C01810=1014.320,152.108,374.636,166.710,56.034,160.285
C01811=1014.316,151.858,374.655,166.706,56.046,160.287
C01812=1014.312,151.609,374.675,166.703,56.058,160.288
C01813=1014.308,151.360,374.694,166.700,56.069,160.290
C01814=1014.304,151.110,374.713,166.697,56.080,160.291
C01815=1014.299,150.861,374.732,166.693,56.091,160.293
C01816=1014.295,150.612,374.751,166.690,56.103,160.294
C01817=1014.291,150.363,374.771,166.686,56.115,160.296
C01818=1014.287,150.113,374.789,166.683,56.126,160.297
C01819=1014.283,149.864,374.809,166.680,56.138,160.299
C01820=1014.279,149.615,374.827,166.676,56.149,160.300
C01821=1014.275,149.366,374.847,166.673,56.160,160.302
C01822=1014.270,149.116,374.865,166.670,56.172,160.303
C01823=1014.266,148.867,374.884,166.667,56.183,160.305
C01824=1014.262,148.618,374.903,166.663,56.194,160.306
C01825=1014.257,148.369,374.923,166.659,56.206,160.308
C01826=1014.253,148.119,374.941,166.656,56.218,160.309
C01827=1014.249,147.870,374.961,166.654,56.229,160.311
C01828=1014.245,147.621,374.979,166.650,56.240,160.312
C01829=1014.241,147.372,374.999,166.646,56.252,160.314
C01830=1014.237,147.122,375.017,166.643,56.263,160.315
C01831=1014.233,146.873,375.036,166.640,56.275,160.317
C01832=1014.229,146.624,375.056,166.636,56.286,160.318
C01833=1014.224,146.374,375.074,166.633,56.297,160.320
C01834=1014.220,146.126,375.093,166.630,56.309,160.321
C01835=1014.216,145.876,375.112,166.627,56.321,160.323
C01836=1014.212,145.627,375.130,166.623,56.332,160.324
C01837=1014.208,145.378,375.150,166.620,56.343,160.326
C01838=1014.204,145.128,375.169,166.617,56.355,160.327
C01839=1014.199,144.879,375.186,166.614,56.366,160.329
C01840=1014.195,144.630,375.205,166.610,56.378,160.330
C01841=1014.191,144.381,375.225,166.607,56.389,160.332
C01842=1014.186,144.131,375.243,166.603,56.401,160.333
C01843=1014.182,143.882,375.262,166.601,56.412,160.335
C01844=1014.178,143.633,375.279,166.598,56.424,160.336
C01845=1014.174,143.384,375.299,166.594,56.435,160.338
C01846=1014.170,143.134,375.318,166.591,56.446,160.339
C01847=1014.165,142.885,375.336,166.587,56.458,160.341
C01848=1014.161,142.636,375.354,166.585,56.469,160.342
C01849=1014.157,142.386,375.373,166.582,56.481,160.344
C01850=1014.153,142.137,375.391,166.578,56.492,160.345
C01851=1014.148,141.888,375.411,166.575,56.504,160.347
C01852=1014.145,141.639,375.429,166.572,56.515,160.349
C01853=1014.140,141.390,375.447,166.568,56.526,160.350
C01854=1014.136,141.140,375.466,166.565,56.538,160.351
C01855=1014.132,140.890,375.485,166.562,56.550,160.353
C01856=1014.128,140.642,375.502,166.560,56.561,160.355
C01857=1014.124,140.392,375.521,166.556,56.572,160.356
C01858=1014.119,140.143,375.541,166.553,56.584,160.357
C01859=1014.115,139.894,375.558,166.550,56.595,160.359
C01860=1014.111,139.645,375.577,166.546,56.606,160.360
C01861=1014.107,139.395,375.596,166.543,56.618,160.362
C01862=1014.102,139.146,375.614,166.540,56.629,160.364
C01863=1014.098,138.866,375.635,166.537,56.642,160.365
C01864=1014.094,138.586,375.656,166.533,56.654,160.367
C01865=1014.088,138.306,375.677,166.529,56.667,160.368
C01866=1014.085,138.026,375.697,166.526,56.680,160.370
C01867=1014.080,137.776,375.715,166.523,56.691,160.372
C01868=1014.076,137.527,375.734,166.520,56.703,160.373
C01869=1014.072,137.278,375.752,166.516,56.714,160.375
C01870=1014.068,137.028,375.770,166.514,56.725,160.376
C01871=1014.063,136.779,375.789,166.511,56.737,160.378
C01872=1014.060,136.530,375.807,166.507,56.748,160.379
C01873=1014.055,136.281,375.825,166.505,56.759,160.381
C01874=1014.051,136.031,375.844,166.502,56.771,160.383
C01875=1014.047,135.782,375.862,166.498,56.782,160.384
C01876=1014.043,135.533,375.881,166.496,56.794,160.386
C01877=1014.038,135.283,375.899,166.493,56.805,160.387
C01878=1014.034,135.034,375.917,166.489,56.817,160.388
C01879=1014.030,134.784,375.935,166.487,56.828,160.390
C01880=1014.025,134.535,375.953,166.483,56.839,160.391
C01881=1014.022,134.286,375.971,166.480,56.851,160.393
C01882=1014.017,134.037,375.989,166.478,56.862,160.395
C01883=1014.013,133.788,376.007,166.474,56.873,160.396
C01884=1014.009,133.538,376.026,166.471,56.885,160.398
C01885=1014.004,133.288,376.043,166.469,56.896,160.399
C01886=1014.001,133.039,376.062,166.465,56.907,160.401
C01887=1013.996,132.790,376.080,166.463,56.919,160.402
C01888=1013.992,132.541,376.098,166.459,56.930,160.404
C01889=1013.988,132.291,376.116,166.456,56.942,160.405
C01890=1013.984,132.043,376.133,166.454,56.953,160.407
C01891=1013.979,131.793,376.152,166.450,56.964,160.408
C01892=1013.975,131.544,376.170,166.448,56.975,160.410
C01893=1013.971,131.295,376.188,166.444,56.987,160.411
C01894=1013.967,131.045,376.206,166.441,56.998,160.413
C01895=1013.963,130.796,376.224,166.438,57.009,160.414
C01896=1013.958,130.547,376.242,166.435,57.021,160.416
C01897=1013.955,130.298,376.261,166.432,57.032,160.418
C01898=1013.950,130.048,376.278,166.429,57.043,160.419
C01899=1013.946,129.798,376.297,166.427,57.054,160.421
C01900=1013.942,129.549,376.315,166.424,57.066,160.422
C01901=1013.938,129.299,376.332,166.421,57.077,160.424
C01902=1013.933,129.051,376.350,166.418,57.088,160.425
C01903=1013.929,128.801,376.367,166.415,57.100,160.427
C01904=1013.925,128.552,376.385,166.412,57.111,160.428
C01905=1013.921,128.302,376.403,166.409,57.123,160.430
C01906=1013.917,128.053,376.421,166.406,57.135,160.431
C01907=1013.912,127.803,376.438,166.403,57.145,160.433
C01908=1013.908,127.555,376.456,166.400,57.157,160.435
C01909=1013.904,127.305,376.474,166.397,57.168,160.436
C01910=1013.899,127.056,376.491,166.394,57.180,160.438
C01911=1013.895,126.806,376.509,166.391,57.192,160.439
C01912=1013.891,126.557,376.526,166.389,57.202,160.441
C01913=1013.886,126.307,376.544,166.386,57.214,160.442
C01914=1013.882,126.058,376.561,166.383,57.225,160.444
C01915=1013.878,125.809,376.579,166.380,57.237,160.445
C01916=1013.874,125.559,376.596,166.377,57.247,160.447
C01917=1013.869,125.310,376.614,166.374,57.259,160.448
C01918=1013.865,125.061,376.632,166.371,57.270,160.450
C01919=1013.861,124.811,376.649,166.369,57.282,160.452
C01920=1013.856,124.562,376.667,166.366,57.294,160.453
C01921=1013.852,124.312,376.684,166.363,57.304,160.455
C01922=1013.848,124.064,376.702,166.360,57.316,160.456
C01923=1013.843,123.814,376.719,166.357,57.327,160.458
C01924=1013.839,123.564,376.737,166.354,57.338,160.459
C01925=1013.835,123.315,376.755,166.352,57.350,160.461
C01926=1013.831,123.066,376.772,166.348,57.361,160.462
C01927=1013.826,122.786,376.791,166.346,57.373,160.464
C01928=1013.821,122.506,376.811,166.342,57.386,160.466
C01929=1013.817,122.226,376.831,166.340,57.399,160.468
C01930=1013.812,121.946,376.850,166.336,57.411,160.469
C01931=1013.807,121.697,376.868,166.334,57.423,160.471
C01932=1013.803,121.447,376.885,166.330,57.434,160.472
C01933=1013.799,121.197,376.903,166.328,57.445,160.474
C01934=1013.795,120.949,376.920,166.326,57.456,160.475
C01935=1013.791,120.699,376.937,166.322,57.467,160.477
C01936=1013.786,120.449,376.955,166.319,57.478,160.478
C01937=1013.782,120.201,376.973,166.316,57.490,160.480
C01938=1013.778,119.952,376.990,166.314,57.501,160.481
C01939=1013.774,119.702,377.007,166.311,57.511,160.483
C01940=1013.770,119.453,377.025,166.308,57.523,160.485
C01941=1013.765,119.203,377.042,166.306,57.534,160.486
C01942=1013.761,118.954,377.060,166.302,57.545,160.487
C01943=1013.757,118.704,377.077,166.300,57.557,160.489
C01944=1013.753,118.455,377.095,166.298,57.568,160.491
C01945=1013.749,118.206,377.112,166.294,57.579,160.492
C01946=1013.745,117.956,377.129,166.292,57.589,160.493
C01947=1013.740,117.707,377.146,166.290,57.601,160.495
C01948=1013.736,117.458,377.164,166.286,57.612,160.497
C01949=1013.732,117.209,377.181,166.284,57.623,160.498
C01950=1013.728,116.959,377.199,166.281,57.634,160.500
C01951=1013.724,116.709,377.216,166.279,57.645,160.501
C01952=1013.720,116.461,377.234,166.276,57.656,160.503
C01953=1013.715,116.211,377.251,166.273,57.667,160.504
C01954=1013.712,115.961,377.269,166.271,57.678,160.506
C01955=1013.708,115.712,377.286,166.267,57.689,160.507
C01956=1013.704,115.462,377.303,166.265,57.700,160.509
C01957=1013.700,115.213,377.321,166.263,57.711,160.510
C01958=1013.696,114.964,377.338,166.261,57.722,160.512
C01959=1013.691,114.714,377.356,166.257,57.733,160.513
C01960=1013.687,114.465,377.373,166.255,57.744,160.515
C01961=1013.683,114.215,377.390,166.252,57.755,160.516
C01962=1013.680,113.966,377.407,166.250,57.766,160.518
C01963=1013.675,113.717,377.425,166.247,57.777,160.519
C01964=1013.671,113.468,377.442,166.244,57.788,160.521
C01965=1013.667,113.218,377.459,166.241,57.799,160.522
C01966=1013.663,112.969,377.476,166.239,57.809,160.524
C01967=1013.659,112.719,377.494,166.237,57.821,160.526
C01968=1013.655,112.470,377.511,166.235,57.832,160.527
C01969=1013.651,112.221,377.528,166.232,57.843,160.529
C01970=1013.647,111.972,377.546,166.229,57.854,160.530
C01971=1013.642,111.722,377.563,166.226,57.865,160.532
C01972=1013.638,111.473,377.579,166.224,57.875,160.533
C01973=1013.634,111.224,377.597,166.221,57.886,160.535
C01974=1013.630,110.973,377.613,166.218,57.897,160.536
C01975=1013.625,110.724,377.630,166.215,57.908,160.537
C01976=1013.621,110.475,377.647,166.213,57.919,160.539
C01977=1013.617,110.226,377.664,166.211,57.930,160.541
C01978=1013.613,109.977,377.680,166.208,57.941,160.542
C01979=1013.608,109.727,377.698,166.205,57.953,160.544
C01980=1013.604,109.477,377.715,166.203,57.964,160.545
C01981=1013.600,109.228,377.732,166.201,57.974,160.547
C01982=1013.596,108.979,377.749,166.198,57.985,160.548
C01983=1013.591,108.729,377.766,166.196,57.996,160.550
C01984=1013.587,108.480,377.782,166.192,58.007,160.551
C01985=1013.583,108.230,377.799,166.190,58.018,160.553
C01986=1013.579,107.981,377.815,166.188,58.029,160.554
C01987=1013.575,107.732,377.832,166.185,58.040,160.556
C01988=1013.570,107.482,377.849,166.183,58.051,160.557
C01989=1013.566,107.233,377.866,166.179,58.062,160.559
C01990=1013.561,106.984,377.882,166.177,58.073,160.560
C01991=1013.557,106.704,377.901,166.175,58.085,160.562
C01992=1013.552,106.423,377.919,166.172,58.097,160.564
C01993=1013.547,106.144,377.939,166.169,58.109,160.566
C01994=1013.542,105.864,377.957,166.166,58.121,160.567
C01995=1013.538,105.615,377.974,166.163,58.133,160.569
C01996=1013.534,105.365,377.990,166.161,58.144,160.570
C01997=1013.530,105.116,378.007,166.158,58.154,160.572
C01998=1013.525,104.867,378.024,166.156,58.165,160.573
C01999=1013.522,104.617,378.040,166.154,58.176,160.575
C02000=1013.517,104.367,378.057,166.151,58.187,160.576
C02001=1013.513,104.118,378.074,166.149,58.198,160.578
C02002=1013.508,103.869,378.090,166.147,58.209,160.579
C02003=1013.505,103.619,378.107,166.144,58.220,160.581
C02004=1013.500,103.370,378.123,166.141,58.231,160.582
C02005=1013.496,103.121,378.140,166.139,58.242,160.584
C02006=1013.492,102.871,378.156,166.136,58.253,160.586
C02007=1013.488,102.622,378.173,166.133,58.263,160.587
C02008=1013.483,102.372,378.189,166.131,58.274,160.588
C02009=1013.479,102.123,378.206,166.129,58.285,160.590
C02010=1013.475,101.874,378.223,166.126,58.295,160.591
C02011=1013.471,101.624,378.239,166.124,58.306,160.593
C02012=1013.467,101.374,378.256,166.122,58.317,160.595
C02013=1013.463,101.125,378.273,166.119,58.327,160.596
C02014=1013.459,100.876,378.289,166.117,58.338,160.597
C02015=1013.454,100.627,378.306,166.114,58.349,160.599
C02016=1013.450,100.377,378.323,166.112,58.360,160.601
C02017=1013.446,100.128,378.338,166.109,58.370,160.602
C02018=1013.442,99.878,378.356,166.107,58.381,160.603
C02019=1013.437,99.628,378.372,166.106,58.391,160.605
C02020=1013.434,99.379,378.389,166.103,58.402,160.607
C02021=1013.429,99.130,378.405,166.100,58.412,160.608
C02022=1013.425,98.880,378.422,166.098,58.423,160.610
C02023=1013.421,98.631,378.438,166.096,58.434,160.611
C02024=1013.416,98.382,378.454,166.093,58.444,160.612
C02025=1013.412,98.132,378.470,166.091,58.455,160.614
C02026=1013.408,97.883,378.487,166.088,58.466,160.616
C02027=1013.404,97.633,378.502,166.086,58.477,160.617
C02028=1013.399,97.384,378.519,166.084,58.488,160.619
C02029=1013.395,97.135,378.535,166.081,58.498,160.620
C02030=1013.391,96.885,378.551,166.079,58.509,160.622
C02031=1013.387,96.636,378.568,166.077,58.520,160.623
C02032=1013.383,96.386,378.583,166.074,58.530,160.624
C02033=1013.378,96.137,378.599,166.072,58.541,160.626
C02034=1013.374,95.888,378.616,166.069,58.552,160.628
C02035=1013.370,95.638,378.632,166.067,58.563,160.629
C02036=1013.366,95.388,378.648,166.064,58.573,160.630
C02037=1013.361,95.139,378.664,166.062,58.584,160.632
C02038=1013.357,94.890,378.680,166.059,58.594,160.633
C02039=1013.353,94.640,378.696,166.058,58.605,160.635
C02040=1013.349,94.391,378.713,166.056,58.616,160.637
C02041=1013.344,94.141,378.729,166.053,58.626,160.638
C02042=1013.340,93.892,378.744,166.051,58.637,160.639
C02043=1013.335,93.643,378.761,166.048,58.647,160.641
C02044=1013.331,93.393,378.777,166.046,58.658,160.642
C02045=1013.328,93.143,378.793,166.043,58.669,160.644
C02046=1013.323,92.894,378.809,166.042,58.679,160.645
C02047=1013.319,92.645,378.825,166.040,58.689,160.647
C02048=1013.314,92.395,378.841,166.037,58.700,160.648
C02049=1013.310,92.146,378.857,166.035,58.711,160.650
C02050=1013.306,91.896,378.874,166.032,58.721,160.651
C02051=1013.302,91.647,378.890,166.031,58.731,160.653
C02052=1013.298,91.397,378.905,166.028,58.742,160.654
C02053=1013.293,91.148,378.922,166.025,58.752,160.655
C02054=1013.289,90.899,378.938,166.023,58.763,160.657
C02055=1013.285,90.619,378.956,166.021,58.774,160.659
C02056=1013.279,90.339,378.974,166.018,58.786,160.660
C02057=1013.275,90.060,378.992,166.015,58.798,160.662
C02058=1013.270,89.781,379.010,166.013,58.809,160.664
C02059=1013.266,89.531,379.025,166.011,58.819,160.665
C02060=1013.262,89.282,379.042,166.008,58.830,160.667
C02061=1013.258,89.032,379.058,166.007,58.840,160.668
C02062=1013.254,88.782,379.073,166.004,58.850,160.669
C02063=1013.249,88.533,379.090,166.002,58.861,160.671
C02064=1013.245,88.284,379.106,166.000,58.871,160.673
C02065=1013.240,88.034,379.121,165.998,58.882,160.674
C02066=1013.236,87.785,379.137,165.995,58.892,160.675
C02067=1013.232,87.535,379.153,165.992,58.902,160.677
C02068=1013.227,87.286,379.169,165.991,58.913,160.679
C02069=1013.223,87.036,379.184,165.989,58.923,160.680
C02070=1013.219,86.787,379.200,165.986,58.934,160.681
C02071=1013.214,86.538,379.215,165.984,58.944,160.683
C02072=1013.210,86.288,379.231,165.982,58.954,160.684
C02073=1013.206,86.039,379.247,165.980,58.965,160.686
C02074=1013.201,85.789,379.262,165.977,58.975,160.687
C02075=1013.197,85.539,379.278,165.975,58.985,160.689
C02076=1013.193,85.290,379.294,165.973,58.996,160.690
C02077=1013.189,85.040,379.309,165.971,59.006,160.692
C02078=1013.185,84.790,379.325,165.969,59.016,160.693
C02079=1013.180,84.542,379.340,165.966,59.026,160.694
C02080=1013.176,84.292,379.355,165.964,59.037,160.696
C02081=1013.172,84.042,379.371,165.962,59.047,160.697
C02082=1013.167,83.793,379.387,165.960,59.057,160.699
C02083=1013.163,83.543,379.403,165.958,59.067,160.700
C02084=1013.159,83.294,379.418,165.955,59.077,160.702
C02085=1013.154,83.044,379.434,165.954,59.087,160.703
C02086=1013.151,82.795,379.450,165.952,59.098,160.705
C02087=1013.146,82.546,379.465,165.949,59.108,160.706
C02088=1013.141,82.296,379.480,165.947,59.118,160.708
C02089=1013.137,82.047,379.496,165.945,59.128,160.709
C02090=1013.133,81.797,379.512,165.943,59.138,160.710
C02091=1013.129,81.548,379.527,165.940,59.149,160.712
C02092=1013.125,81.298,379.542,165.939,59.158,160.713
C02093=1013.121,81.049,379.558,165.936,59.169,160.714
C02094=1013.116,80.799,379.574,165.934,59.178,160.716
C02095=1013.111,80.550,379.589,165.932,59.189,160.717
C02096=1013.107,80.300,379.605,165.930,59.199,160.719
C02097=1013.103,80.051,379.620,165.927,59.209,160.720
C02098=1013.099,79.802,379.636,165.926,59.219,160.722
C02099=1013.095,79.551,379.651,165.923,59.229,160.723
C02100=1013.091,79.302,379.667,165.921,59.239,160.724
C02101=1013.086,79.052,379.683,165.920,59.249,160.726
C02102=1013.083,78.803,379.698,165.917,59.259,160.727
C02103=1013.078,78.554,379.713,165.915,59.269,160.729
C02104=1013.073,78.305,379.729,165.913,59.279,160.730
C02105=1013.069,78.055,379.745,165.911,59.289,160.732
C02106=1013.066,77.806,379.760,165.910,59.299,160.733
C02107=1013.061,77.556,379.775,165.906,59.308,160.734
C02108=1013.057,77.306,379.791,165.905,59.318,160.736
C02109=1013.053,77.057,379.807,165.903,59.328,160.737
C02110=1013.049,76.807,379.822,165.900,59.338,160.739
C02111=1013.044,76.558,379.837,165.899,59.348,160.740
C02112=1013.040,76.308,379.852,165.897,59.358,160.742
C02113=1013.036,76.059,379.868,165.894,59.367,160.743
C02114=1013.031,75.809,379.883,165.892,59.377,160.744
C02115=1013.027,75.560,379.898,165.891,59.387,160.746
C02116=1013.023,75.311,379.914,165.888,59.397,160.747
C02117=1013.018,75.061,379.928,165.887,59.407,160.749
C02118=1013.014,74.811,379.944,165.884,59.418,160.750
C02119=1013.010,74.572,379.958,165.882,59.427,160.751
C02120=1013.006,74.331,379.973,165.880,59.436,160.752
C02121=1013.002,74.092,379.987,165.878,59.446,160.754
C02122=1012.997,73.852,380.002,165.876,59.455,160.755
C02123=1012.994,73.612,380.017,165.874,59.465,160.757
C02124=1012.989,73.372,380.031,165.872,59.474,160.758
C02125=1012.985,73.133,380.045,165.870,59.484,160.759
C02126=1012.981,72.892,380.060,165.868,59.493,160.761
C02127=1012.977,72.643,380.075,165.867,59.503,160.762
C02128=1012.973,72.393,380.090,165.865,59.512,160.763
C02129=1012.968,72.144,380.105,165.862,59.522,160.765
C02130=1012.964,71.895,380.121,165.860,59.532,160.766
C02131=1012.959,71.645,380.135,165.858,59.541,160.767
C02132=1012.955,71.396,380.151,165.857,59.551,160.769
C02133=1012.951,71.147,380.165,165.854,59.560,160.770
C02134=1012.947,70.897,380.181,165.852,59.570,160.771
C02135=1012.943,70.647,380.196,165.850,59.580,160.773
C02136=1012.938,70.398,380.211,165.848,59.589,160.774
C02137=1012.934,70.148,380.226,165.847,59.599,160.776
C02138=1012.929,69.899,380.241,165.844,59.608,160.777
C02139=1012.926,69.649,380.256,165.843,59.618,160.779
C02140=1012.921,69.400,380.271,165.840,59.628,160.780
C02141=1012.917,69.150,380.286,165.838,59.638,160.781
C02142=1012.912,68.901,380.301,165.836,59.647,160.782
C02143=1012.908,68.651,380.316,165.835,59.657,160.784
C02144=1012.903,68.402,380.331,165.832,59.666,160.785
C02145=1012.900,68.152,380.346,165.830,59.675,160.786
C02146=1012.895,67.903,380.361,165.829,59.685,160.788
C02147=1012.891,67.653,380.376,165.827,59.694,160.789
C02148=1012.887,67.404,380.390,165.825,59.704,160.791
C02149=1012.882,67.154,380.406,165.823,59.713,160.792
C02150=1012.878,66.904,380.420,165.821,59.723,160.793
C02151=1012.874,66.655,380.435,165.818,59.733,160.794
C02152=1012.869,66.405,380.450,165.816,59.742,160.796
C02153=1012.865,66.156,380.464,165.815,59.752,160.797
C02154=1012.861,65.906,380.479,165.812,59.761,160.798
C02155=1012.856,65.657,380.494,165.810,59.770,160.800
C02156=1012.853,65.407,380.509,165.809,59.780,160.801
C02157=1012.848,65.157,380.523,165.807,59.789,160.802
C02158=1012.843,64.909,380.538,165.805,59.798,160.804
C02159=1012.839,64.659,380.553,165.803,59.808,160.805
C02160=1012.835,64.409,380.568,165.801,59.817,160.806
C02161=1012.830,64.160,380.583,165.799,59.826,160.808
C02162=1012.826,63.910,380.598,165.797,59.836,160.809
C02163=1012.822,63.661,380.612,165.795,59.845,160.811
C02164=1012.817,63.411,380.626,165.793,59.855,160.812
C02165=1012.813,63.161,380.642,165.791,59.864,160.813
C02166=1012.809,62.912,380.656,165.790,59.873,160.814
C02167=1012.804,62.662,380.671,165.788,59.882,160.816
C02168=1012.801,62.413,380.685,165.786,59.891,160.817
C02169=1012.796,62.163,380.700,165.784,59.901,160.818
C02170=1012.791,61.913,380.714,165.782,59.910,160.820
C02171=1012.787,61.664,380.728,165.780,59.919,160.821
C02172=1012.782,61.414,380.743,165.778,59.928,160.822
C02173=1012.778,61.165,380.757,165.777,59.938,160.824
C02174=1012.773,60.915,380.772,165.775,59.947,160.825
C02175=1012.769,60.666,380.786,165.773,59.957,160.826
C02176=1012.764,60.416,380.800,165.770,59.966,160.827
C02177=1012.760,60.167,380.815,165.768,59.975,160.829
C02178=1012.755,59.917,380.829,165.766,59.984,160.830
C02179=1012.732,71.816,379.715,165.827,59.747,160.800
C02180=1012.736,72.066,379.701,165.829,59.737,160.799
C02181=1012.741,72.316,379.685,165.831,59.728,160.797
C02182=1012.745,72.565,379.671,165.833,59.719,160.796
C02183=1012.749,72.814,379.655,165.834,59.709,160.795
C02184=1012.753,73.059,379.641,165.837,59.700,160.793
C02185=1012.757,73.305,379.627,165.839,59.691,160.792
C02186=1012.762,73.551,379.612,165.840,59.681,160.791
C02187=1012.765,73.796,379.597,165.842,59.672,160.789
C02188=1012.770,74.042,379.582,165.844,59.662,160.788
C02189=1012.774,74.286,379.567,165.846,59.653,160.787
C02190=1012.778,74.532,379.552,165.848,59.644,160.785
C02191=1012.783,74.778,379.537,165.851,59.633,160.784
C02192=1012.787,75.026,379.522,165.853,59.624,160.783
C02193=1012.791,75.276,379.507,165.854,59.614,160.781
C02194=1012.796,75.526,379.492,165.856,59.604,160.780
C02195=1012.799,75.775,379.477,165.858,59.595,160.778
C02196=1012.803,76.025,379.461,165.861,59.585,160.777
C02197=1012.809,76.274,379.446,165.863,59.576,160.776
C02198=1012.812,76.524,379.431,165.864,59.566,160.774
C02199=1012.816,76.773,379.416,165.866,59.556,160.773
C02200=1012.820,77.024,379.401,165.868,59.547,160.772
C02201=1012.825,77.273,379.385,165.871,59.537,160.770
C02202=1012.829,77.522,379.370,165.873,59.528,160.769
C02203=1012.833,77.771,379.354,165.874,59.518,160.767
C02204=1012.837,78.021,379.339,165.876,59.508,160.766
C02205=1012.842,78.271,379.323,165.879,59.498,160.765
C02206=1012.845,78.520,379.308,165.881,59.488,160.763
C02207=1012.850,78.769,379.292,165.882,59.478,160.762
C02208=1012.854,79.020,379.277,165.884,59.469,160.761
C02209=1012.858,79.268,379.262,165.887,59.459,160.759
C02210=1012.862,79.518,379.247,165.889,59.449,160.758
C02211=1012.867,79.767,379.231,165.890,59.439,160.756
C02212=1012.871,80.017,379.215,165.894,59.430,160.755
C02213=1012.874,80.266,379.200,165.895,59.420,160.754
C02214=1012.879,80.516,379.185,165.897,59.410,160.752
C02215=1012.883,80.766,379.169,165.899,59.400,160.751
C02216=1012.887,81.015,379.153,165.901,59.390,160.749
C02217=1012.891,81.264,379.138,165.902,59.380,160.748
C02218=1012.896,81.513,379.122,165.906,59.371,160.747
C02219=1012.900,81.764,379.107,165.907,59.361,160.745
C02220=1012.904,82.013,379.092,165.910,59.350,160.744
C02221=1012.908,82.262,379.076,165.911,59.341,160.742
C02222=1012.912,82.512,379.060,165.913,59.331,160.741
C02223=1012.917,82.761,379.045,165.916,59.320,160.740
C02224=1012.921,83.011,379.029,165.917,59.311,160.738
C02225=1012.925,83.261,379.014,165.920,59.300,160.737
C02226=1012.929,83.509,378.999,165.922,59.290,160.735
C02227=1012.934,83.759,378.983,165.924,59.280,160.734
C02228=1012.938,84.009,378.968,165.926,59.270,160.732
C02229=1012.942,84.258,378.952,165.928,59.260,160.731
C02230=1012.947,84.508,378.936,165.930,59.250,160.729
C02231=1012.950,84.757,378.921,165.933,59.240,160.728
C02232=1012.954,85.007,378.906,165.934,59.230,160.727
C02233=1012.959,85.256,378.890,165.937,59.220,160.725
C02234=1012.964,85.506,378.875,165.939,59.210,160.724
C02235=1012.968,85.755,378.859,165.941,59.200,160.722
C02236=1012.972,86.005,378.843,165.942,59.189,160.721
C02237=1012.976,86.254,378.828,165.945,59.179,160.719
C02238=1012.980,86.503,378.812,165.948,59.169,160.718
C02239=1012.985,86.753,378.796,165.949,59.159,160.716
C02240=1012.989,87.002,378.780,165.952,59.149,160.715
C02241=1012.993,87.252,378.765,165.954,59.139,160.714
C02242=1012.997,87.502,378.749,165.956,59.128,160.712
C02243=1013.002,87.750,378.734,165.958,59.117,160.711
C02244=1013.006,88.000,378.718,165.960,59.108,160.709
C02245=1013.010,88.250,378.703,165.963,59.097,160.708
C02246=1013.015,88.500,378.687,165.965,59.086,160.706
C02247=1013.019,88.749,378.672,165.966,59.077,160.705
C02248=1013.023,88.998,378.655,165.969,59.066,160.703
C02249=1013.027,89.248,378.639,165.972,59.056,160.702
C02250=1013.031,89.498,378.623,165.974,59.046,160.701
C02251=1013.035,89.746,378.608,165.976,59.035,160.699
C02252=1013.041,90.026,378.590,165.978,59.024,160.697
C02253=1013.045,90.306,378.571,165.981,59.013,160.696
C02254=1013.049,90.585,378.554,165.982,59.001,160.694
C02255=1013.054,90.864,378.536,165.986,58.990,160.693
C02256=1013.058,91.114,378.520,165.988,58.979,160.691
C02257=1013.062,91.363,378.504,165.989,58.969,160.689
C02258=1013.067,91.613,378.488,165.992,58.959,160.688
C02259=1013.070,91.862,378.471,165.995,58.948,160.687
C02260=1013.075,92.112,378.455,165.996,58.938,160.685
C02261=1013.078,92.360,378.440,165.999,58.928,160.684
C02262=1013.083,92.610,378.424,166.001,58.917,160.682
C02263=1013.087,92.860,378.408,166.004,58.906,160.681
C02264=1013.091,93.109,378.391,166.005,58.897,160.679
C02265=1013.095,93.358,378.376,166.008,58.886,160.678
C02266=1013.100,93.608,378.360,166.010,58.876,160.676
C02267=1013.104,93.858,378.344,166.013,58.865,160.675
C02268=1013.108,94.107,378.328,166.014,58.855,160.673
C02269=1013.112,94.356,378.311,166.017,58.845,160.672
C02270=1013.116,94.606,378.295,166.019,58.834,160.670
C02271=1013.121,94.856,378.280,166.022,58.823,160.669
C02272=1013.125,95.105,378.263,166.024,58.812,160.668
C02273=1013.130,95.354,378.247,166.026,58.803,160.666
C02274=1013.133,95.604,378.231,166.028,58.792,160.664
C02275=1013.137,95.854,378.215,166.030,58.781,160.663
C02276=1013.142,96.103,378.199,166.033,58.771,160.662
C02277=1013.146,96.352,378.183,166.035,58.760,160.660
C02278=1013.151,96.602,378.167,166.038,58.749,160.659
C02279=1013.154,96.850,378.151,166.040,58.739,160.657
C02280=1013.158,97.100,378.135,166.042,58.729,160.656
C02281=1013.163,97.349,378.119,166.044,58.718,160.654
C02282=1013.167,97.599,378.103,166.047,58.708,160.653
C02283=1013.171,97.848,378.087,166.049,58.697,160.651
C02284=1013.175,98.098,378.070,166.051,58.686,160.650
C02285=1013.179,98.347,378.055,166.054,58.675,160.648
C02286=1013.184,98.596,378.038,166.056,58.665,160.647
C02287=1013.187,98.846,378.022,166.058,58.654,160.645
C02288=1013.193,99.096,378.005,166.061,58.643,160.644
C02289=1013.196,99.346,377.989,166.063,58.632,160.642
C02290=1013.201,99.595,377.972,166.066,58.622,160.641
C02291=1013.204,99.845,377.956,166.067,58.612,160.639
C02292=1013.209,100.094,377.939,166.069,58.601,160.638
C02293=1013.213,100.344,377.923,166.072,58.591,160.636
C02294=1013.217,100.592,377.906,166.074,58.580,160.635
C02295=1013.221,100.842,377.890,166.077,58.570,160.633
C02296=1013.225,101.091,377.874,166.079,58.559,160.632
C02297=1013.229,101.341,377.857,166.082,58.548,160.630
C02298=1013.234,101.590,377.841,166.084,58.537,160.629
C02299=1013.237,101.839,377.824,166.087,58.527,160.627
C02300=1013.242,102.089,377.808,166.089,58.516,160.626
C02301=1013.246,102.338,377.791,166.091,58.505,160.624
C02302=1013.250,102.588,377.775,166.094,58.495,160.623
C02303=1013.254,102.837,377.758,166.096,58.484,160.621
C02304=1013.258,103.087,377.742,166.099,58.473,160.620
C02305=1013.262,103.336,377.725,166.101,58.462,160.618
C02306=1013.267,103.585,377.709,166.104,58.452,160.617
C02307=1013.270,103.835,377.692,166.106,58.441,160.615
C02308=1013.275,104.084,377.676,166.108,58.430,160.614
C02309=1013.278,104.334,377.659,166.111,58.419,160.612
C02310=1013.284,104.583,377.643,166.113,58.408,160.611
C02311=1013.287,104.833,377.625,166.115,58.397,160.609
C02312=1013.292,105.082,377.610,166.118,58.387,160.608
C02313=1013.296,105.331,377.593,166.120,58.376,160.606
C02314=1013.300,105.580,377.576,166.123,58.365,160.605
C02315=1013.304,105.830,377.560,166.125,58.355,160.603
C02316=1013.309,106.110,377.540,166.129,58.342,160.602
C02317=1013.314,106.390,377.522,166.131,58.330,160.600
C02318=1013.318,106.669,377.504,166.133,58.317,160.598
C02319=1013.323,106.949,377.486,166.136,58.305,160.596
C02320=1013.327,107.198,377.469,166.138,58.294,160.595
C02321=1013.332,107.447,377.452,166.141,58.283,160.593
C02322=1013.335,107.697,377.436,166.143,58.273,160.592
C02323=1013.340,107.947,377.418,166.146,58.261,160.590
C02324=1013.344,108.196,377.402,166.149,58.250,160.589
C02325=1013.348,108.446,377.385,166.151,58.240,160.587
C02326=1013.352,108.695,377.369,166.153,58.229,160.585
C02327=1013.356,108.944,377.352,166.156,58.218,160.584
C02328=1013.361,109.193,377.335,166.158,58.207,160.582
C02329=1013.364,109.443,377.319,166.161,58.196,160.581
C02330=1013.369,109.693,377.302,166.164,58.185,160.579
C02331=1013.374,109.942,377.285,166.166,58.174,160.578
C02332=1013.377,110.191,377.268,166.168,58.163,160.576
C02333=1013.381,110.440,377.251,166.171,58.152,160.575
C02334=1013.385,110.690,377.234,166.174,58.141,160.573
C02335=1013.390,110.939,377.218,166.177,58.130,160.572
C02336=1013.394,111.189,377.201,166.179,58.119,160.570
C02337=1013.398,111.439,377.184,166.181,58.108,160.569
C02338=1013.402,111.688,377.167,166.184,58.098,160.567
C02339=1013.406,111.937,377.150,166.187,58.086,160.566
C02340=1013.410,112.186,377.133,166.189,58.075,160.564
C02341=1013.415,112.436,377.115,166.192,58.065,160.563
C02342=1013.419,112.685,377.098,166.194,58.054,160.561
C02343=1013.422,112.935,377.081,166.196,58.043,160.560
C02344=1013.426,113.184,377.064,166.199,58.032,160.558
C02345=1013.430,113.433,377.047,166.202,58.021,160.557
C02346=1013.435,113.683,377.030,166.205,58.010,160.555
C02347=1013.439,113.932,377.012,166.207,57.999,160.554
C02348=1013.443,114.181,376.995,166.209,57.988,160.552
C02349=1013.447,114.430,376.978,166.212,57.977,160.551
C02350=1013.451,114.680,376.960,166.215,57.966,160.549
C02351=1013.455,114.930,376.943,166.218,57.955,160.548
C02352=1013.459,115.179,376.926,166.220,57.945,160.546
C02353=1013.463,115.428,376.909,166.222,57.934,160.545
C02354=1013.467,115.678,376.892,166.226,57.923,160.543
C02355=1013.471,115.927,376.875,166.228,57.911,160.541
C02356=1013.475,116.176,376.857,166.230,57.900,160.540
C02357=1013.479,116.425,376.840,166.233,57.889,160.538
C02358=1013.484,116.675,376.822,166.236,57.878,160.537
C02359=1013.487,116.924,376.805,166.238,57.867,160.536
C02360=1013.491,117.174,376.788,166.241,57.857,160.534
C02361=1013.495,117.423,376.771,166.243,57.846,160.532
C02362=1013.500,117.673,376.754,166.246,57.834,160.531
C02363=1013.504,117.922,376.736,166.249,57.823,160.529
C02364=1013.508,118.171,376.719,166.251,57.812,160.528
C02365=1013.511,118.421,376.701,166.255,57.801,160.526
C02366=1013.515,118.670,376.684,166.256,57.789,160.525
C02367=1013.519,118.920,376.666,166.260,57.778,160.523
C02368=1013.523,119.168,376.649,166.262,57.767,160.522
C02369=1013.528,119.418,376.631,166.265,57.757,160.520
C02370=1013.532,119.668,376.614,166.268,57.745,160.519
C02371=1013.536,119.917,376.597,166.270,57.734,160.517
C02372=1013.540,120.167,376.580,166.273,57.723,160.516
C02373=1013.544,120.415,376.562,166.276,57.712,160.514
C02374=1013.548,120.665,376.545,166.278,57.700,160.512
C02375=1013.553,120.915,376.527,166.282,57.689,160.511
C02376=1013.556,121.164,376.510,166.284,57.678,160.510
C02377=1013.561,121.413,376.492,166.287,57.666,160.508
C02378=1013.565,121.663,376.475,166.290,57.656,160.506
C02379=1013.569,121.912,376.458,166.291,57.644,160.505
C02380=1013.574,122.191,376.439,166.295,57.632,160.503
C02381=1013.578,122.471,376.419,166.298,57.619,160.501
C02382=1013.584,122.752,376.400,166.302,57.607,160.500
C02383=1013.588,123.032,376.380,166.305,57.594,160.498
C02384=1013.592,123.280,376.362,166.307,57.582,160.496
C02385=1013.597,123.530,376.345,166.311,57.571,160.495
C02386=1013.600,123.780,376.327,166.313,57.560,160.493
C02387=1013.605,124.028,376.310,166.316,57.548,160.492
C02388=1013.609,124.278,376.292,166.319,57.538,160.490
C02389=1013.613,124.527,376.275,166.322,57.526,160.489
C02390=1013.617,124.777,376.258,166.324,57.515,160.487
C02391=1013.622,125.026,376.240,166.327,57.503,160.485
C02392=1013.626,125.275,376.223,166.330,57.492,160.484
C02393=1013.630,125.525,376.205,166.333,57.480,160.482
C02394=1013.634,125.774,376.188,166.335,57.470,160.481
C02395=1013.639,126.024,376.170,166.338,57.458,160.479
C02396=1013.643,126.273,376.152,166.342,57.447,160.478
C02397=1013.647,126.522,376.135,166.344,57.435,160.476
C02398=1013.651,126.772,376.118,166.347,57.423,160.474
C02399=1013.655,127.020,376.100,166.349,57.412,160.473
C02400=1013.660,127.270,376.083,166.352,57.401,160.471
C02401=1013.664,127.520,376.066,166.356,57.389,160.470
C02402=1013.668,127.769,376.047,166.358,57.378,160.468
C02403=1013.672,128.018,376.030,166.361,57.366,160.467
C02404=1013.677,128.268,376.012,166.365,57.355,160.465
C02405=1013.681,128.517,375.995,166.367,57.343,160.464
C02406=1013.685,128.766,375.978,166.370,57.332,160.462
C02407=1013.690,129.016,375.960,166.373,57.320,160.461
C02408=1013.694,129.265,375.943,166.375,57.309,160.459
C02409=1013.698,129.515,375.924,166.379,57.298,160.458
C02410=1013.702,129.765,375.907,166.381,57.286,160.456
C02411=1013.705,130.013,375.888,166.384,57.275,160.454
C02412=1013.710,130.263,375.870,166.388,57.263,160.453
C02413=1013.714,130.512,375.853,166.390,57.253,160.451
C02414=1013.718,130.762,375.834,166.393,57.241,160.450
C02415=1013.722,131.010,375.816,166.396,57.230,160.448
C02416=1013.727,131.260,375.799,166.399,57.218,160.447
C02417=1013.730,131.509,375.781,166.403,57.207,160.445
C02418=1013.735,131.759,375.762,166.405,57.196,160.444
C02419=1013.738,132.008,375.745,166.408,57.185,160.442
C02420=1013.743,132.258,375.727,166.410,57.173,160.440
C02421=1013.747,132.506,375.709,166.413,57.161,160.439
C02422=1013.751,132.756,375.690,166.417,57.150,160.438
C02423=1013.755,133.005,375.673,166.419,57.139,160.436
C02424=1013.760,133.255,375.655,166.423,57.128,160.435
C02425=1013.763,133.503,375.636,166.426,57.116,160.433
C02426=1013.768,133.753,375.619,166.428,57.104,160.431
C02427=1013.771,134.002,375.600,166.432,57.093,160.430
C02428=1013.776,134.252,375.582,166.435,57.081,160.428
C02429=1013.780,134.500,375.565,166.437,57.070,160.427
C02430=1013.784,134.751,375.546,166.440,57.059,160.425
C02431=1013.789,135.000,375.528,166.444,57.047,160.424
C02432=1013.792,135.249,375.510,166.447,57.035,160.422
C02433=1013.797,135.498,375.492,166.449,57.025,160.421
C02434=1013.800,135.747,375.473,166.453,57.013,160.419
C02435=1013.805,135.997,375.456,166.456,57.001,160.417
C02436=1013.809,136.246,375.438,166.458,56.990,160.416
C02437=1013.813,136.496,375.419,166.461,56.979,160.414
C02438=1013.818,136.745,375.401,166.465,56.967,160.413
C02439=1013.821,136.994,375.383,166.468,56.956,160.411
C02440=1013.826,137.243,375.365,166.470,56.944,160.410
C02441=1013.829,137.492,375.346,166.474,56.932,160.408
C02442=1013.834,137.742,375.329,166.477,56.921,160.407
C02443=1013.838,137.992,375.310,166.481,56.910,160.405
C02444=1013.843,138.271,375.289,166.483,56.897,160.403
C02445=1013.847,138.551,375.268,166.487,56.884,160.402
C02446=1013.851,138.831,375.248,166.490,56.871,160.400
C02447=1013.857,139.111,375.227,166.494,56.858,160.398
C02448=1013.861,139.361,375.208,166.497,56.848,160.397
C02449=1013.864,139.609,375.190,166.500,56.836,160.395
C02450=1013.869,139.859,375.172,166.503,56.824,160.394
C02451=1013.872,140.108,375.153,166.506,56.812,160.392
C02452=1013.876,140.357,375.135,166.509,56.802,160.391
C02453=1013.881,140.607,375.116,166.512,56.790,160.389
C02454=1013.885,140.856,375.098,166.516,56.778,160.388
C02455=1013.889,141.105,375.080,166.519,56.767,160.386
C02456=1013.893,141.355,375.061,166.522,56.755,160.385
C02457=1013.897,141.604,375.043,166.525,56.744,160.383
C02458=1013.902,141.853,375.025,166.528,56.732,160.381
C02459=1013.906,142.103,375.006,166.532,56.721,160.380
C02460=1013.909,142.352,374.987,166.535,56.709,160.379
C02461=1013.914,142.601,374.969,166.538,56.698,160.377
C02462=1013.918,142.850,374.950,166.540,56.686,160.375
C02463=1013.922,143.100,374.931,166.544,56.674,160.374
C02464=1013.926,143.348,374.913,166.547,56.663,160.372
C02465=1013.930,143.598,374.894,166.551,56.652,160.371
C02466=1013.934,143.848,374.876,166.554,56.640,160.369
C02467=1013.939,144.096,374.858,166.557,56.628,160.368
C02468=1013.943,144.346,374.839,166.560,56.616,160.366
C02469=1013.947,144.596,374.820,166.564,56.605,160.365
C02470=1013.952,144.844,374.802,166.566,56.594,160.363
C02471=1013.955,145.093,374.783,166.570,56.582,160.362
C02472=1013.959,145.343,374.764,166.573,56.571,160.360
C02473=1013.963,145.593,374.746,166.576,56.559,160.358
C02474=1013.968,145.841,374.727,166.580,56.548,160.357
C02475=1013.972,146.090,374.708,166.583,56.536,160.356
C02476=1013.976,146.340,374.690,166.587,56.524,160.354
C02477=1013.980,146.590,374.671,166.589,56.513,160.352
C02478=1013.984,146.839,374.651,166.592,56.501,160.351
C02479=1013.988,147.088,374.633,166.596,56.490,160.350
C02480=1013.992,147.337,374.614,166.599,56.479,160.348
C02481=1013.997,147.586,374.595,166.603,56.467,160.346
C02482=1014.001,147.836,374.577,166.606,56.455,160.345
C02483=1014.005,148.085,374.558,166.609,56.444,160.343
C02484=1014.009,148.334,374.539,166.612,56.432,160.342
C02485=1014.013,148.583,374.520,166.615,56.421,160.340
C02486=1014.017,148.833,374.501,166.619,56.410,160.339
C02487=1014.021,149.082,374.482,166.622,56.398,160.337
C02488=1014.025,149.332,374.463,166.625,56.386,160.336
C02489=1014.029,149.580,374.444,166.629,56.374,160.334
C02490=1014.033,149.830,374.425,166.632,56.364,160.333
C02491=1014.037,150.079,374.406,166.636,56.352,160.331
C02492=1014.041,150.329,374.387,166.639,56.340,160.330
C02493=1014.046,150.578,374.367,166.642,56.328,160.328
C02494=1014.050,150.827,374.349,166.646,56.317,160.327
C02495=1014.054,151.075,374.330,166.649,56.305,160.325
C02496=1014.058,151.325,374.311,166.652,56.293,160.324
C02497=1014.063,151.574,374.292,166.656,56.282,160.322
C02498=1014.067,151.824,374.273,166.660,56.271,160.321
C02499=1014.071,152.073,374.254,166.663,56.259,160.319
C02500=1014.075,152.322,374.235,166.666,56.247,160.318
C02501=1014.079,152.571,374.215,166.670,56.236,160.316
C02502=1014.083,152.820,374.197,166.673,56.224,160.315
C02503=1014.087,153.069,374.178,166.676,56.212,160.313
C02504=1014.091,153.319,374.159,166.679,56.201,160.311
C02505=1014.095,153.568,374.139,166.682,56.189,160.310
C02506=1014.099,153.817,374.119,166.686,56.179,160.309
C02507=1014.103,154.067,374.101,166.689,56.167,160.307
C02508=1014.108,154.347,374.078,166.694,56.154,160.306
C02509=1014.113,154.627,374.057,166.698,56.140,160.304
C02510=1014.118,154.907,374.036,166.702,56.127,160.302
C02511=1014.122,155.187,374.014,166.706,56.115,160.301
C02512=1014.126,155.436,373.995,166.709,56.103,160.299
C02513=1014.131,155.685,373.975,166.712,56.091,160.297
C02514=1014.134,155.934,373.957,166.716,56.080,160.296
C02515=1014.139,156.183,373.937,166.719,56.068,160.294
C02516=1014.143,156.432,373.918,166.723,56.056,160.293
C02517=1014.146,156.682,373.899,166.726,56.045,160.291
C02518=1014.151,156.931,373.879,166.729,56.033,160.290
C02519=1014.155,157.180,373.860,166.733,56.021,160.288
C02520=1014.159,157.429,373.840,166.736,56.010,160.287
C02521=1014.163,157.679,373.821,166.740,55.998,160.285
C02522=1014.168,157.928,373.802,166.743,55.987,160.284
C02523=1014.172,158.177,373.782,166.747,55.976,160.282
C02524=1014.176,158.426,373.762,166.751,55.964,160.281
C02525=1014.180,158.675,373.743,166.754,55.952,160.279
C02526=1014.184,158.925,373.723,166.757,55.941,160.278
C02527=1014.187,159.174,373.703,166.761,55.929,160.276
C02528=1014.192,159.423,373.683,166.765,55.918,160.275
C02529=1014.195,159.672,373.663,166.768,55.907,160.274
C02530=1014.200,159.921,373.644,166.772,55.895,160.272
C02531=1014.203,160.171,373.624,166.775,55.884,160.271
C02532=1014.208,160.420,373.604,166.779,55.873,160.269
C02533=1014.211,160.669,373.584,166.783,55.861,160.268
C02534=1014.215,160.918,373.564,166.786,55.849,160.266
C02535=1014.219,161.168,373.545,166.790,55.838,160.265
C02536=1014.223,161.417,373.525,166.794,55.827,160.264
C02537=1014.227,161.666,373.505,166.797,55.815,160.262
C02538=1014.231,161.915,373.485,166.801,55.804,160.261
C02539=1014.235,162.164,373.466,166.804,55.792,160.259
C02540=1014.240,162.414,373.444,166.808,55.781,160.257
C02541=1014.243,162.663,373.424,166.811,55.769,160.256
C02542=1014.247,162.912,373.405,166.815,55.758,160.255
C02543=1014.251,163.162,373.385,166.819,55.747,160.253
C02544=1014.255,163.411,373.365,166.822,55.735,160.252
C02545=1014.259,163.660,373.345,166.826,55.723,160.250
C02546=1014.264,163.908,373.325,166.829,55.712,160.249
C02547=1014.267,164.158,373.305,166.833,55.700,160.247
C02548=1014.271,164.407,373.285,166.837,55.689,160.246
C02549=1014.275,164.656,373.265,166.840,55.678,160.244
C02550=1014.279,164.905,373.245,166.845,55.666,160.243
C02551=1014.283,165.154,373.226,166.848,55.654,160.242
C02552=1014.287,165.403,373.205,166.852,55.643,160.240
C02553=1014.292,165.653,373.185,166.855,55.631,160.239
C02554=1014.296,165.902,373.165,166.859,55.620,160.237
C02555=1014.299,166.152,373.145,166.863,55.608,160.236
C02556=1014.304,166.400,373.125,166.866,55.597,160.234
C02557=1014.308,166.649,373.105,166.870,55.586,160.233
C02558=1014.312,166.898,373.085,166.874,55.574,160.231
C02559=1014.316,167.148,373.065,166.878,55.562,160.230
C02560=1014.319,167.397,373.045,166.882,55.551,160.228
C02561=1014.324,167.646,373.025,166.885,55.539,160.227
C02562=1014.328,167.896,373.005,166.889,55.528,160.225
C02563=1014.333,168.144,372.984,166.893,55.516,160.224
C02564=1014.336,168.393,372.964,166.896,55.505,160.222
C02565=1014.341,168.642,372.945,166.901,55.493,160.221
C02566=1014.345,168.892,372.924,166.904,55.481,160.220
C02567=1014.349,169.141,372.904,166.908,55.470,160.218
C02568=1014.353,169.390,372.884,166.912,55.458,160.217
C02569=1014.357,169.639,372.863,166.915,55.447,160.215
C02570=1014.361,169.888,372.844,166.920,55.435,160.214
C02571=1014.366,170.138,372.824,166.923,55.423,160.212
C02572=1014.370,170.418,372.801,166.927,55.411,160.211
C02573=1014.375,170.697,372.778,166.933,55.397,160.209
C02574=1014.379,170.976,372.755,166.936,55.384,160.207
C02575=1014.384,171.256,372.733,166.940,55.372,160.206
C02576=1014.388,171.505,372.713,166.945,55.360,160.204
C02577=1014.393,171.755,372.692,166.949,55.348,160.203
C02578=1014.397,172.004,372.672,166.952,55.337,160.201
C02579=1014.401,172.253,372.652,166.956,55.325,160.200
C02580=1014.405,172.502,372.632,166.960,55.313,160.199
C02581=1014.409,172.751,372.611,166.964,55.302,160.197
C02582=1014.414,173.000,372.592,166.968,55.290,160.196
C02583=1014.417,173.249,372.571,166.972,55.278,160.194
C02584=1014.422,173.499,372.550,166.976,55.267,160.193
C02585=1014.426,173.748,372.531,166.980,55.255,160.191
C02586=1014.430,173.997,372.510,166.984,55.244,160.190
C02587=1014.435,174.246,372.490,166.988,55.232,160.188
C02588=1014.439,174.495,372.469,166.992,55.221,160.187
C02589=1014.443,174.744,372.450,166.996,55.209,160.186
C02590=1014.447,174.993,372.429,167.000,55.197,160.184
C02591=1014.452,175.243,372.409,167.003,55.185,160.182
C02592=1014.456,175.491,372.389,167.008,55.173,160.181
C02593=1014.461,175.741,372.367,167.011,55.162,160.180
C02594=1014.465,175.990,372.348,167.015,55.150,160.178
C02595=1014.469,176.239,372.327,167.020,55.138,160.177
C02596=1014.473,176.489,372.307,167.024,55.127,160.175
C02597=1014.478,176.737,372.287,167.028,55.115,160.174
C02598=1014.481,176.986,372.266,167.032,55.104,160.173
C02599=1014.487,177.236,372.246,167.036,55.092,160.171
C02600=1014.491,177.484,372.225,167.040,55.080,160.170
C02601=1014.495,177.734,372.205,167.044,55.069,160.168
C02602=1014.499,177.983,372.185,167.049,55.057,160.167
C02603=1014.503,178.232,372.164,167.052,55.045,160.165
C02604=1014.508,178.481,372.144,167.056,55.034,160.164
C02605=1014.512,178.730,372.123,167.060,55.022,160.162
C02606=1014.516,178.980,372.103,167.064,55.010,160.161
C02607=1014.521,179.228,372.082,167.069,54.998,160.160
C02608=1014.526,179.478,372.061,167.073,54.987,160.158
C02609=1014.530,179.726,372.041,167.077,54.975,160.157
C02610=1014.534,179.976,372.021,167.081,54.964,160.155
C02611=1014.538,180.225,372.000,167.085,54.951,160.154
C02612=1014.543,180.474,371.980,167.089,54.940,160.152
C02613=1014.547,180.724,371.959,167.094,54.928,160.151
C02614=1014.552,180.972,371.939,167.097,54.917,160.149
C02615=1014.556,181.221,371.918,167.102,54.905,160.148
C02616=1014.560,181.470,371.897,167.106,54.893,160.147
C02617=1014.565,181.720,371.877,167.111,54.882,160.145
C02618=1014.569,181.969,371.856,167.114,54.870,160.144
C02619=1014.573,182.218,371.834,167.118,54.859,160.142
C02620=1014.577,182.468,371.812,167.122,54.847,160.141
C02621=1014.581,182.716,371.792,167.127,54.836,160.140
C02622=1014.585,182.965,371.771,167.131,54.825,160.138
C02623=1014.589,183.215,371.749,167.135,54.814,160.137
C02624=1014.593,183.463,371.728,167.140,54.802,160.135
C02625=1014.597,183.713,371.707,167.143,54.790,160.134
C02626=1014.601,183.962,371.686,167.147,54.779,160.133
C02627=1014.605,184.211,371.664,167.152,54.768,160.131
C02628=1014.609,184.460,371.643,167.156,54.757,160.130
C02629=1014.614,184.709,371.622,167.160,54.745,160.129
C02630=1014.618,184.958,371.601,167.165,54.733,160.127
C02631=1014.621,185.207,371.579,167.169,54.722,160.126
C02632=1014.626,185.456,371.558,167.172,54.711,160.124
C02633=1014.630,185.705,371.537,167.177,54.699,160.123
C02634=1014.635,185.954,371.516,167.181,54.688,160.122
C02635=1014.638,186.203,371.494,167.186,54.676,160.120
C02636=1014.643,186.483,371.470,167.190,54.663,160.119
C02637=1014.647,186.762,371.446,167.196,54.650,160.117
C02638=1014.652,187.042,371.422,167.200,54.638,160.116
C02639=1014.657,187.321,371.398,167.205,54.625,160.114
C02640=1014.661,187.571,371.377,167.209,54.614,160.113
C02641=1014.665,187.819,371.356,167.214,54.602,160.111
C02642=1014.669,188.069,371.334,167.218,54.591,160.110
C02643=1014.674,188.318,371.313,167.223,54.579,160.109
C02644=1014.678,188.566,371.291,167.226,54.568,160.107
C02645=1014.682,188.815,371.270,167.231,54.556,160.106
C02646=1014.686,189.065,371.249,167.236,54.545,160.105
C02647=1014.690,189.313,371.227,167.239,54.534,160.103
C02648=1014.695,189.563,371.206,167.244,54.522,160.102
C02649=1014.698,189.811,371.184,167.248,54.511,160.100
C02650=1014.703,190.061,371.163,167.253,54.499,160.099
C02651=1014.707,190.310,371.141,167.257,54.488,160.098
C02652=1014.712,190.559,371.120,167.262,54.476,160.096
C02653=1014.715,190.808,371.098,167.266,54.465,160.095
C02654=1014.720,191.057,371.076,167.270,54.453,160.093
C02655=1014.725,191.306,371.055,167.274,54.442,160.092
C02656=1014.729,191.554,371.034,167.279,54.430,160.091
C02657=1014.733,191.804,371.012,167.284,54.418,160.089
C02658=1014.737,192.053,370.991,167.288,54.408,160.088
C02659=1014.741,192.302,370.969,167.293,54.396,160.087
C02660=1014.745,192.551,370.948,167.297,54.385,160.085
C02661=1014.750,192.800,370.926,167.302,54.373,160.084
C02662=1014.755,193.050,370.905,167.306,54.362,160.083
C02663=1014.759,193.298,370.883,167.311,54.350,160.081
C02664=1014.763,193.547,370.861,167.315,54.339,160.080
C02665=1014.767,193.796,370.839,167.320,54.327,160.079
C02666=1014.772,194.045,370.818,167.325,54.316,160.077
C02667=1014.776,194.294,370.797,167.329,54.304,160.076
C02668=1014.780,194.543,370.774,167.334,54.293,160.074
C02669=1014.785,194.792,370.753,167.337,54.281,160.073
C02670=1014.790,195.041,370.731,167.342,54.270,160.072
C02671=1014.793,195.291,370.710,167.347,54.258,160.070
C02672=1014.798,195.540,370.688,167.351,54.247,160.069
C02673=1014.802,195.788,370.666,167.356,54.235,160.068
C02674=1014.807,196.037,370.645,167.362,54.224,160.067
C02675=1014.811,196.286,370.623,167.365,54.213,160.065
C02676=1014.816,196.535,370.601,167.370,54.201,160.064
C02677=1014.820,196.785,370.580,167.375,54.190,160.062
C02678=1014.824,197.034,370.557,167.379,54.178,160.061
C02679=1014.829,197.282,370.536,167.384,54.167,160.060
C02680=1014.833,197.531,370.515,167.389,54.155,160.058
C02681=1014.838,197.780,370.493,167.393,54.144,160.057
C02682=1014.842,198.029,370.470,167.398,54.132,160.056
C02683=1014.847,198.279,370.449,167.403,54.121,160.054
C02684=1014.851,198.528,370.427,167.407,54.109,160.053
C02685=1014.856,198.777,370.405,167.412,54.098,160.052
C02686=1014.860,199.025,370.383,167.417,54.086,160.050
C02687=1014.864,199.275,370.361,167.421,54.075,160.049
C02688=1014.869,199.524,370.339,167.426,54.063,160.047
C02689=1014.872,199.772,370.317,167.431,54.052,160.046
C02690=1014.877,200.022,370.295,167.435,54.041,160.045
C02691=1014.881,200.270,370.273,167.440,54.029,160.044
C02692=1014.885,200.520,370.250,167.444,54.018,160.042
C02693=1014.890,200.769,370.228,167.449,54.007,160.041
C02694=1014.894,201.017,370.206,167.455,53.996,160.040
C02695=1014.898,201.267,370.184,167.459,53.985,160.038
C02696=1014.903,201.516,370.161,167.464,53.973,160.037
C02697=1014.907,201.765,370.139,167.469,53.961,160.036
C02698=1014.911,202.014,370.117,167.473,53.951,160.035
C02699=1014.916,202.262,370.094,167.478,53.939,160.033
C02700=1014.935,203.369,369.995,167.998,54.006,160.161
C02701=1014.941,203.601,369.973,168.002,53.997,160.160
C02702=1014.945,203.833,369.951,168.006,53.987,160.159
C02703=1014.950,204.064,369.928,168.010,53.978,160.158
C02704=1014.956,204.297,369.906,168.014,53.968,160.157
C02705=1014.960,204.529,369.883,168.018,53.959,160.155
C02706=1014.966,204.760,369.861,168.022,53.949,160.154
C02707=1014.971,204.993,369.839,168.026,53.940,160.153
C02708=1014.976,205.225,369.816,168.031,53.930,160.152
C02709=1014.981,205.473,369.792,168.034,53.920,160.151
C02710=1014.986,205.722,369.768,168.039,53.910,160.149
C02711=1014.992,205.972,369.744,168.043,53.900,160.148
C02712=1014.997,206.220,369.720,168.048,53.890,160.147
C02713=1015.002,206.469,369.695,168.053,53.880,160.146
C02714=1015.008,206.717,369.671,168.056,53.870,160.145
C02715=1015.013,206.966,369.647,168.060,53.859,160.143
C02716=1015.018,207.215,369.623,168.065,53.850,160.142
C02717=1015.024,207.463,369.598,168.070,53.839,160.141
C02718=1015.030,207.712,369.574,168.074,53.830,160.140
C02719=1015.035,207.961,369.550,168.078,53.819,160.138
C02720=1015.040,208.210,369.525,168.083,53.810,160.137
C02721=1015.045,208.458,369.501,168.086,53.800,160.136
C02722=1015.051,208.707,369.477,168.091,53.790,160.135
C02723=1015.057,208.956,369.452,168.096,53.780,160.134
C02724=1015.062,209.205,369.428,168.100,53.770,160.133
C02725=1015.067,209.453,369.404,168.104,53.760,160.131
C02726=1015.073,209.702,369.379,168.109,53.751,160.130
C02727=1015.078,209.951,369.354,168.113,53.741,160.129
C02728=1015.083,210.200,369.330,168.117,53.731,160.128
C02729=1015.088,210.449,369.306,168.122,53.721,160.127
C02730=1015.094,210.697,369.281,168.126,53.711,160.125
C02731=1015.099,210.946,369.257,168.131,53.701,160.124
C02732=1015.104,211.195,369.231,168.135,53.692,160.123
C02733=1015.110,211.443,369.207,168.139,53.682,160.122
C02734=1015.115,211.692,369.183,168.143,53.673,160.121
C02735=1015.121,211.941,369.158,168.148,53.663,160.120
C02736=1015.125,212.190,369.133,168.153,53.653,160.119
C02737=1015.131,212.438,369.108,168.157,53.644,160.117
C02738=1015.136,212.687,369.084,168.162,53.634,160.116
C02739=1015.142,212.936,369.059,168.165,53.625,160.115
C02740=1015.147,213.185,369.034,168.170,53.615,160.114
C02741=1015.152,213.433,369.010,168.174,53.606,160.113
C02742=1015.158,213.682,368.985,168.179,53.596,160.112
C02743=1015.164,213.931,368.961,168.183,53.587,160.111
C02744=1015.169,214.179,368.936,168.188,53.576,160.109
C02745=1015.174,214.428,368.910,168.191,53.567,160.108
C02746=1015.180,214.677,368.886,168.196,53.557,160.107
C02747=1015.186,214.926,368.862,168.200,53.548,160.106
C02748=1015.191,215.174,368.837,168.205,53.538,160.105
C02749=1015.196,215.423,368.812,168.209,53.529,160.104
C02750=1015.202,215.672,368.787,168.214,53.519,160.103
C02751=1015.207,215.920,368.762,168.218,53.510,160.102
C02752=1015.213,216.169,368.738,168.223,53.500,160.101
C02753=1015.218,216.418,368.713,168.227,53.491,160.099
C02754=1015.223,216.666,368.688,168.232,53.482,160.099
C02755=1015.229,216.916,368.663,168.236,53.473,160.097
C02756=1015.235,217.164,368.638,168.241,53.463,160.096
C02757=1015.240,217.413,368.613,168.245,53.454,160.095
C02758=1015.246,217.661,368.588,168.250,53.444,160.094
C02759=1015.251,217.910,368.564,168.254,53.435,160.093
C02760=1015.256,218.159,368.538,168.258,53.426,160.092
C02761=1015.262,218.402,368.514,168.263,53.417,160.091
C02762=1015.267,218.646,368.489,168.267,53.407,160.090
C02763=1015.272,218.889,368.464,168.272,53.399,160.089
C02764=1015.278,219.133,368.440,168.276,53.390,160.088
C02765=1015.283,219.377,368.415,168.280,53.381,160.087
C02766=1015.288,219.620,368.390,168.284,53.372,160.086
C02767=1015.293,219.864,368.365,168.289,53.363,160.085
C02768=1015.298,220.107,368.341,168.294,53.353,160.084
C02769=1015.304,220.356,368.315,168.298,53.345,160.083
C02770=1015.309,220.605,368.291,168.302,53.336,160.082
C02771=1015.315,220.854,368.265,168.306,53.327,160.081
C02772=1015.320,221.102,368.240,168.311,53.317,160.080
C02773=1015.326,221.351,368.214,168.316,53.309,160.079
C02774=1015.331,221.599,368.190,168.320,53.300,160.077
C02775=1015.336,221.848,368.164,168.325,53.290,160.076
C02776=1015.342,222.097,368.138,168.329,53.281,160.076
C02777=1015.348,222.345,368.113,168.333,53.272,160.074
C02778=1015.353,222.595,368.088,168.338,53.264,160.073
C02779=1015.358,222.843,368.063,168.343,53.254,160.072
C02780=1015.364,223.092,368.037,168.347,53.245,160.071
C02781=1015.369,223.340,368.012,168.351,53.237,160.071
C02782=1015.375,223.589,367.986,168.355,53.228,160.069
C02783=1015.381,223.838,367.961,168.361,53.219,160.069
C02784=1015.386,224.086,367.936,168.365,53.210,160.067
C02785=1015.392,224.335,367.911,168.369,53.201,160.066
C02786=1015.397,224.583,367.885,168.373,53.192,160.065
C02787=1015.402,224.832,367.859,168.379,53.183,160.064
C02788=1015.408,225.081,367.834,168.383,53.174,160.064
C02789=1015.413,225.329,367.808,168.387,53.165,160.062
C02790=1015.419,225.578,367.784,168.392,53.157,160.061
C02791=1015.425,225.827,367.758,168.396,53.148,160.060
C02792=1015.430,226.075,367.733,168.401,53.138,160.059
C02793=1015.436,226.324,367.707,168.406,53.130,160.058
C02794=1015.441,226.573,367.681,168.410,53.121,160.058
C02795=1015.446,226.822,367.655,168.415,53.113,160.057
C02796=1015.453,227.070,367.629,168.419,53.104,160.056
C02797=1015.457,227.318,367.604,168.423,53.095,160.055
C02798=1015.463,227.567,367.578,168.428,53.087,160.054
C02799=1015.468,227.816,367.552,168.433,53.078,160.053
C02800=1015.474,228.065,367.526,168.438,53.069,160.052
C02801=1015.479,228.313,367.501,168.442,53.061,160.051
C02802=1015.485,228.562,367.475,168.446,53.052,160.050
C02803=1015.490,228.811,367.449,168.451,53.044,160.049
C02804=1015.496,229.058,367.423,168.455,53.035,160.048
C02805=1015.501,229.307,367.397,168.460,53.027,160.047
C02806=1015.507,229.556,367.371,168.464,53.018,160.046
C02807=1015.512,229.804,367.346,168.469,53.010,160.045
C02808=1015.518,230.053,367.319,168.473,53.001,160.044
C02809=1015.523,230.302,367.293,168.478,52.993,160.043
C02810=1015.529,230.551,367.267,168.482,52.984,160.043
C02811=1015.534,230.799,367.242,168.487,52.976,160.042
C02812=1015.539,231.047,367.215,168.491,52.967,160.041
C02813=1015.545,231.296,367.189,168.496,52.959,160.040
C02814=1015.550,231.545,367.163,168.500,52.950,160.039
C02815=1015.556,231.793,367.137,168.505,52.942,160.038
C02816=1015.561,232.042,367.111,168.510,52.934,160.037
C02817=1015.567,232.290,367.084,168.514,52.925,160.036
C02818=1015.572,232.539,367.058,168.519,52.917,160.035
C02819=1015.578,232.788,367.032,168.523,52.908,160.034
C02820=1015.583,233.036,367.006,168.528,52.900,160.033
C02821=1015.589,233.275,366.982,168.533,52.892,160.033
C02822=1015.594,233.515,366.956,168.537,52.884,160.032
C02823=1015.599,233.755,366.931,168.541,52.876,160.031
C02824=1015.605,233.994,366.906,168.546,52.868,160.030
C02825=1015.610,234.234,366.880,168.551,52.860,160.029
C02826=1015.615,234.474,366.855,168.554,52.852,160.028
C02827=1015.621,234.712,366.830,168.559,52.844,160.028
C02828=1015.626,234.952,366.805,168.564,52.836,160.027
C02829=1015.631,235.200,366.778,168.569,52.828,160.026
C02830=1015.637,235.449,366.752,168.572,52.820,160.025
C02831=1015.643,235.697,366.726,168.577,52.812,160.024
C02832=1015.648,235.946,366.700,168.582,52.803,160.023
C02833=1015.654,236.195,366.673,168.586,52.795,160.022
C02834=1015.660,236.443,366.646,168.591,52.787,160.022
C02835=1015.665,236.692,366.621,168.596,52.779,160.021
C02836=1015.671,236.940,366.594,168.601,52.771,160.020
C02837=1015.676,237.189,366.568,168.605,52.762,160.019
C02838=1015.682,237.437,366.542,168.610,52.754,160.018
C02839=1015.687,237.685,366.515,168.615,52.746,160.017
C02840=1015.693,237.934,366.489,168.619,52.738,160.016
C02841=1015.699,238.183,366.462,168.623,52.730,160.016
C02842=1015.704,238.431,366.436,168.628,52.722,160.015
C02843=1015.710,238.679,366.409,168.633,52.714,160.014
C02844=1015.716,238.928,366.383,168.638,52.706,160.013
C02845=1015.721,239.177,366.356,168.642,52.698,160.012
C02846=1015.726,239.425,366.329,168.647,52.690,160.012
C02847=1015.732,239.674,366.303,168.651,52.682,160.011
C02848=1015.737,239.923,366.275,168.656,52.674,160.010
C02849=1015.743,240.171,366.249,168.661,52.667,160.009
C02850=1015.749,240.419,366.222,168.666,52.659,160.008
C02851=1015.755,240.668,366.195,168.670,52.650,160.008
C02852=1015.759,240.917,366.169,168.674,52.643,160.007
C02853=1015.765,241.165,366.142,168.679,52.635,160.006
C02854=1015.771,241.414,366.116,168.684,52.628,160.005
C02855=1015.776,241.662,366.088,168.689,52.619,160.004
C02856=1015.782,241.911,366.062,168.693,52.612,160.004
C02857=1015.787,242.159,366.035,168.698,52.604,160.003
C02858=1015.792,242.408,366.008,168.703,52.596,160.002
C02859=1015.798,242.656,365.981,168.708,52.589,160.001
C02860=1015.804,242.904,365.954,168.711,52.580,160.000
C02861=1015.809,243.152,365.927,168.716,52.573,160.000
C02862=1015.815,243.401,365.900,168.721,52.565,159.999
C02863=1015.820,243.649,365.873,168.726,52.557,159.998
C02864=1015.825,243.898,365.845,168.730,52.550,159.997
C02865=1015.831,244.146,365.819,168.735,52.542,159.997
C02866=1015.836,244.395,365.791,168.740,52.534,159.996
C02867=1015.842,244.643,365.764,168.744,52.527,159.995
C02868=1015.848,244.892,365.737,168.749,52.519,159.995
C02869=1015.853,245.141,365.709,168.754,52.513,159.994
C02870=1015.859,245.389,365.682,168.759,52.505,159.993
C02871=1015.864,245.637,365.655,168.764,52.497,159.993
C02872=1015.870,245.886,365.628,168.768,52.490,159.992
C02873=1015.875,246.134,365.601,168.773,52.482,159.991
C02874=1015.880,246.382,365.573,168.778,52.474,159.990
C02875=1015.886,246.632,365.546,168.782,52.467,159.989
C02876=1015.891,246.880,365.519,168.787,52.459,159.989
C02877=1015.897,247.128,365.491,168.792,52.452,159.988
C02878=1015.903,247.377,365.464,168.796,52.445,159.987
C02879=1015.908,247.625,365.437,168.801,52.437,159.987
C02880=1015.914,247.873,365.409,168.806,52.430,159.986
C02881=1015.920,248.149,365.379,168.811,52.421,159.985
C02882=1015.926,248.424,365.349,168.816,52.413,159.984
C02883=1015.933,248.700,365.319,168.822,52.405,159.984
C02884=1015.938,248.975,365.288,168.827,52.397,159.983
C02885=1015.945,249.223,365.260,168.832,52.389,159.982
C02886=1015.950,249.472,365.233,168.837,52.382,159.982
C02887=1015.955,249.720,365.205,168.841,52.375,159.981
C02888=1015.961,249.969,365.178,168.846,52.367,159.980
C02889=1015.967,250.217,365.150,168.850,52.360,159.979
C02890=1015.972,250.465,365.124,168.856,52.353,159.979
C02891=1015.978,250.713,365.096,168.861,52.345,159.978
C02892=1015.983,250.963,365.068,168.865,52.338,159.977
C02893=1015.988,251.184,365.043,168.869,52.331,159.977
C02894=1015.994,251.408,365.019,168.874,52.325,159.976
C02895=1015.999,251.630,364.994,168.879,52.319,159.976
C02896=1016.004,251.853,364.970,168.882,52.312,159.975
C02897=1016.009,252.075,364.945,168.887,52.306,159.974
C02898=1016.014,252.298,364.920,168.891,52.299,159.974
C02899=1016.019,252.520,364.896,168.896,52.292,159.973
C02900=1016.024,252.743,364.871,168.900,52.286,159.973
C02901=1016.030,252.991,364.843,168.904,52.279,159.972
C02902=1016.036,253.240,364.816,168.910,52.271,159.971
C02903=1016.041,253.488,364.788,168.914,52.264,159.970
C02904=1016.047,253.737,364.760,168.919,52.257,159.970
C02905=1016.053,253.985,364.733,168.924,52.249,159.969
C02906=1016.058,254.234,364.706,168.929,52.243,159.969
C02907=1016.065,254.482,364.678,168.934,52.235,159.968
C02908=1016.070,254.730,364.650,168.938,52.229,159.967
C02909=1016.076,254.979,364.622,168.944,52.222,159.967
C02910=1016.082,255.227,364.595,168.948,52.214,159.966
C02911=1016.088,255.475,364.567,168.953,52.207,159.966
C02912=1016.093,255.724,364.539,168.958,52.200,159.965
C02913=1016.099,255.972,364.512,168.963,52.193,159.964
C02914=1016.105,256.221,364.484,168.968,52.185,159.963
C02915=1016.111,256.469,364.456,168.972,52.179,159.963
C02916=1016.117,256.718,364.428,168.978,52.172,159.962
C02917=1016.123,256.966,364.400,168.982,52.164,159.962
C02918=1016.129,257.215,364.373,168.987,52.157,159.961
C02919=1016.134,257.463,364.345,168.993,52.150,159.961
C02920=1016.140,257.711,364.317,168.997,52.143,159.960
C02921=1016.146,257.959,364.289,169.002,52.136,159.959
C02922=1016.152,258.208,364.261,169.007,52.130,159.959
C02923=1016.158,258.456,364.234,169.012,52.123,159.958
C02924=1016.164,258.704,364.205,169.016,52.115,159.957
C02925=1016.170,258.952,364.177,169.022,52.108,159.957
C02926=1016.176,259.201,364.150,169.026,52.102,159.956
C02927=1016.182,259.449,364.122,169.032,52.095,159.956
C02928=1016.188,259.697,364.094,169.036,52.087,159.955
C02929=1016.194,259.945,364.066,169.041,52.080,159.954
C02930=1016.199,260.195,364.037,169.046,52.074,159.954
C02931=1016.204,260.443,364.009,169.051,52.067,159.953
C02932=1016.210,260.691,363.981,169.056,52.060,159.953
C02933=1016.216,260.939,363.952,169.060,52.054,159.952
C02934=1016.222,261.188,363.924,169.066,52.047,159.952
C02935=1016.228,261.436,363.895,169.070,52.040,159.951
C02936=1016.233,261.684,363.867,169.076,52.033,159.951
C02937=1016.239,261.932,363.838,169.080,52.027,159.950
C02938=1016.245,262.180,363.810,169.086,52.020,159.950
C02939=1016.251,262.429,363.782,169.091,52.014,159.949
C02940=1016.256,262.678,363.754,169.095,52.007,159.948
C02941=1016.262,262.912,363.727,169.100,52.001,159.948
C02942=1016.268,263.148,363.700,169.105,51.995,159.947
C02943=1016.273,263.383,363.672,169.109,51.988,159.947
C02944=1016.278,263.618,363.646,169.114,51.981,159.946
C02945=1016.284,263.853,363.619,169.119,51.976,159.946
C02946=1016.290,264.088,363.592,169.123,51.969,159.945
C02947=1016.294,264.324,363.565,169.128,51.963,159.945
C02948=1016.300,264.559,363.538,169.133,51.956,159.944
C02949=1016.306,264.807,363.509,169.139,51.950,159.944
C02950=1016.312,265.055,363.481,169.143,51.944,159.943
C02951=1016.318,265.304,363.452,169.149,51.937,159.943
C02952=1016.324,265.552,363.423,169.153,51.930,159.942
C02953=1016.329,265.800,363.395,169.158,51.924,159.942
C02954=1016.335,266.048,363.366,169.164,51.917,159.941
C02955=1016.341,266.297,363.337,169.168,51.911,159.941
C02956=1016.347,266.545,363.308,169.173,51.905,159.940
C02957=1016.353,266.792,363.280,169.179,51.898,159.940
C02958=1016.358,267.042,363.251,169.184,51.892,159.940
C02959=1016.364,267.290,363.222,169.188,51.885,159.939
C02960=1016.370,267.538,363.193,169.194,51.878,159.938
C02961=1016.376,267.786,363.165,169.199,51.873,159.938
C02962=1016.382,268.034,363.136,169.204,51.866,159.938
C02963=1016.387,268.283,363.107,169.209,51.860,159.937
C02964=1016.393,268.531,363.078,169.214,51.853,159.937
C02965=1016.399,268.779,363.049,169.220,51.847,159.936
C02966=1016.405,269.027,363.020,169.224,51.840,159.936
C02967=1016.411,269.276,362.991,169.229,51.834,159.935
C02968=1016.417,269.524,362.962,169.234,51.828,159.935
C02969=1016.423,269.772,362.933,169.240,51.822,159.934
C02970=1016.428,270.020,362.904,169.244,51.815,159.934
C02971=1016.434,270.268,362.875,169.249,51.809,159.933
C02972=1016.440,270.516,362.845,169.255,51.803,159.933
C02973=1016.446,270.765,362.817,169.259,51.796,159.933
C02974=1016.452,271.013,362.788,169.264,51.790,159.932
C02975=1016.457,271.262,362.758,169.270,51.784,159.932
C02976=1016.464,271.510,362.729,169.275,51.778,159.931
C02977=1016.469,271.758,362.700,169.280,51.772,159.931
C02978=1016.475,272.006,362.671,169.285,51.766,159.930
C02979=1016.481,272.254,362.642,169.290,51.759,159.930
C02980=1016.487,272.502,362.612,169.295,51.753,159.930
C02981=1016.493,272.750,362.583,169.300,51.747,159.929
C02982=1016.498,272.999,362.553,169.305,51.741,159.929
C02983=1016.505,273.247,362.524,169.311,51.734,159.928
C02984=1016.510,273.495,362.495,169.316,51.729,159.928
C02985=1016.516,273.744,362.466,169.321,51.723,159.927
C02986=1016.522,273.992,362.436,169.327,51.717,159.927
C02987=1016.528,274.240,362.407,169.332,51.711,159.927
C02988=1016.534,274.489,362.377,169.337,51.705,159.926
C02989=1016.540,274.736,362.348,169.341,51.698,159.926
C02990=1016.546,274.985,362.318,169.347,51.692,159.926
C02991=1016.552,275.233,362.289,169.352,51.686,159.925
C02992=1016.557,275.481,362.259,169.357,51.680,159.925
C02993=1016.563,275.729,362.231,169.362,51.674,159.924
C02994=1016.570,275.976,362.201,169.368,51.668,159.924
C02995=1016.575,276.225,362.171,169.373,51.662,159.924
C02996=1016.581,276.473,362.142,169.378,51.656,159.923
C02997=1016.587,276.721,362.113,169.383,51.651,159.923
C02998=1016.593,276.969,362.082,169.389,51.644,159.923
C02999=1016.598,277.217,362.053,169.394,51.639,159.922
C03000=1016.604,277.465,362.022,169.399,51.633,159.922
C03001=1016.610,277.703,361.994,169.404,51.627,159.922
C03002=1016.616,277.940,361.966,169.409,51.622,159.921
C03003=1016.621,278.178,361.937,169.414,51.616,159.921
C03004=1016.627,278.416,361.908,169.418,51.611,159.921
C03005=1016.633,278.652,361.881,169.423,51.605,159.920
C03006=1016.638,278.890,361.851,169.429,51.600,159.920
C03007=1016.644,279.127,361.823,169.434,51.594,159.920
C03008=1016.649,279.365,361.794,169.439,51.588,159.919
C03009=1016.656,279.612,361.764,169.444,51.583,159.919
C03010=1016.662,279.861,361.735,169.449,51.577,159.919
C03011=1016.667,280.109,361.704,169.455,51.571,159.918
C03012=1016.673,280.357,361.675,169.460,51.565,159.918
C03013=1016.679,280.605,361.645,169.465,51.560,159.918
C03014=1016.686,280.854,361.615,169.470,51.554,159.917
C03015=1016.691,281.102,361.585,169.475,51.548,159.917
C03016=1016.697,281.349,361.554,169.481,51.542,159.917
C03017=1016.703,281.598,361.525,169.487,51.537,159.916
C03018=1016.709,281.845,361.495,169.492,51.531,159.916
C03019=1016.716,282.094,361.464,169.497,51.525,159.916
C03020=1016.722,282.342,361.435,169.502,51.520,159.915
C03021=1016.728,282.590,361.405,169.508,51.514,159.915
C03022=1016.734,282.838,361.374,169.513,51.509,159.915
C03023=1016.739,283.086,361.345,169.518,51.503,159.915
C03024=1016.746,283.334,361.315,169.523,51.497,159.914
C03025=1016.752,283.582,361.284,169.529,51.492,159.914
C03026=1016.758,283.830,361.254,169.535,51.486,159.914
C03027=1016.764,284.079,361.224,169.540,51.480,159.914
C03028=1016.770,284.327,361.194,169.545,51.475,159.913
C03029=1016.776,284.575,361.164,169.551,51.469,159.913
C03030=1016.782,284.822,361.134,169.556,51.464,159.913
C03031=1016.789,285.071,361.103,169.561,51.458,159.912
C03032=1016.794,285.319,361.072,169.567,51.452,159.912
C03033=1016.800,285.567,361.042,169.572,51.447,159.912
C03034=1016.807,285.815,361.011,169.578,51.442,159.912
C03035=1016.812,286.063,360.981,169.583,51.436,159.911
C03036=1016.818,286.311,360.951,169.588,51.431,159.911
C03037=1016.825,286.559,360.920,169.594,51.426,159.911
C03038=1016.830,286.807,360.890,169.600,51.420,159.911
C03039=1016.836,287.055,360.859,169.605,51.414,159.910
C03040=1016.843,287.303,360.829,169.610,51.409,159.910
C03041=1016.849,287.551,360.798,169.615,51.404,159.910
C03042=1016.854,287.799,360.768,169.621,51.398,159.910
C03043=1016.861,288.048,360.737,169.626,51.393,159.909
C03044=1016.867,288.295,360.707,169.632,51.388,159.909
C03045=1016.873,288.543,360.676,169.638,51.383,159.909
C03046=1016.879,288.791,360.645,169.643,51.377,159.909
C03047=1016.885,289.039,360.615,169.648,51.372,159.909
C03048=1016.891,289.287,360.584,169.654,51.366,159.908
C03049=1016.897,289.535,360.554,169.659,51.361,159.908
C03050=1016.904,289.783,360.522,169.665,51.356,159.908
C03051=1016.910,290.031,360.492,169.670,51.351,159.908
C03052=1016.915,290.280,360.461,169.675,51.345,159.907
C03053=1016.921,290.528,360.430,169.681,51.340,159.907
C03054=1016.927,290.775,360.399,169.687,51.335,159.907
C03055=1016.934,291.023,360.368,169.692,51.329,159.907
C03056=1016.940,291.271,360.338,169.698,51.324,159.907
C03057=1016.946,291.519,360.307,169.703,51.319,159.907
C03058=1016.952,291.767,360.276,169.708,51.314,159.906
C03059=1016.959,292.015,360.245,169.714,51.309,159.906
C03060=1016.964,292.263,360.214,169.719,51.304,159.906
C03061=1016.970,292.506,360.184,169.725,51.299,159.906
C03062=1016.977,292.750,360.152,169.730,51.294,159.906
C03063=1016.983,292.993,360.122,169.736,51.289,159.906
C03064=1016.989,293.237,360.091,169.741,51.284,159.905
C03065=1016.994,293.480,360.061,169.747,51.279,159.905
C03066=1017.000,293.724,360.030,169.752,51.274,159.905
C03067=1017.006,293.967,359.999,169.758,51.269,159.905
C03068=1017.011,294.211,359.968,169.763,51.264,159.905
C03069=1017.018,294.459,359.937,169.769,51.259,159.905
C03070=1017.024,294.706,359.905,169.774,51.254,159.905
C03071=1017.030,294.955,359.874,169.780,51.249,159.905
C03072=1017.036,295.203,359.842,169.786,51.245,159.905
C03073=1017.042,295.450,359.811,169.791,51.240,159.904
C03074=1017.048,295.698,359.779,169.797,51.234,159.904
C03075=1017.053,295.946,359.748,169.802,51.230,159.904
C03076=1017.060,296.194,359.717,169.808,51.225,159.904
C03077=1017.066,296.443,359.685,169.814,51.220,159.904
C03078=1017.072,296.690,359.654,169.819,51.215,159.904
C03079=1017.078,296.938,359.622,169.825,51.210,159.904
C03080=1017.085,297.186,359.590,169.831,51.205,159.904
C03081=1017.090,297.434,359.559,169.837,51.200,159.904
C03082=1017.097,297.681,359.527,169.842,51.196,159.904
C03083=1017.103,297.930,359.495,169.848,51.191,159.903
C03084=1017.109,298.177,359.464,169.854,51.186,159.903
C03085=1017.115,298.425,359.432,169.859,51.181,159.903
C03086=1017.121,298.673,359.400,169.865,51.177,159.903
C03087=1017.127,298.920,359.369,169.870,51.171,159.903
C03088=1017.133,299.169,359.337,169.876,51.167,159.903
C03089=1017.140,299.417,359.306,169.882,51.162,159.903
C03090=1017.146,299.665,359.274,169.887,51.157,159.903
C03091=1017.152,299.913,359.242,169.893,51.153,159.903
C03092=1017.158,300.160,359.211,169.899,51.148,159.903
C03093=1017.165,300.408,359.179,169.904,51.143,159.903
C03094=1017.171,300.656,359.147,169.910,51.138,159.903
C03095=1017.178,300.904,359.115,169.917,51.133,159.903
C03096=1017.184,301.152,359.083,169.923,51.129,159.903
C03097=1017.189,301.399,359.051,169.928,51.124,159.902
C03098=1017.196,301.647,359.020,169.934,51.119,159.902
C03099=1017.202,301.895,358.988,169.940,51.115,159.903
C03100=1017.209,302.143,358.956,169.945,51.110,159.902
C03101=1017.215,302.391,358.924,169.951,51.105,159.902
C03102=1017.221,302.639,358.892,169.957,51.101,159.902
C03103=1017.227,302.887,358.860,169.962,51.096,159.902
C03104=1017.234,303.134,358.828,169.968,51.091,159.902
C03105=1017.240,303.382,358.796,169.974,51.087,159.902
C03106=1017.246,303.630,358.764,169.981,51.082,159.902
C03107=1017.253,303.877,358.732,169.986,51.078,159.902
C03108=1017.259,304.126,358.700,169.992,51.073,159.902
C03109=1017.266,304.373,358.669,169.998,51.069,159.902
C03110=1017.272,304.621,358.636,170.003,51.064,159.902
C03111=1017.279,304.869,358.605,170.009,51.059,159.902
C03112=1017.285,305.117,358.572,170.015,51.055,159.902
C03113=1017.292,305.364,358.540,170.021,51.050,159.902
C03114=1017.298,305.613,358.508,170.027,51.046,159.902
C03115=1017.304,305.860,358.476,170.033,51.041,159.902
C03116=1017.311,306.108,358.444,170.039,51.037,159.902
C03117=1017.317,306.356,358.411,170.045,51.032,159.902
C03118=1017.324,306.604,358.380,170.051,51.028,159.902
C03119=1017.330,306.851,358.347,170.057,51.023,159.902
C03120=1017.337,307.100,358.315,170.063,51.019,159.902
C03121=1017.344,307.357,358.282,170.068,51.014,159.902
C03122=1017.351,307.613,358.248,170.075,51.010,159.902
C03123=1017.357,307.870,358.215,170.081,51.005,159.902
C03124=1017.364,308.127,358.181,170.088,51.000,159.902
C03125=1017.370,308.375,358.149,170.094,50.996,159.903
C03126=1017.378,308.623,358.117,170.100,50.992,159.903
C03127=1017.384,308.870,358.084,170.105,50.987,159.903
C03128=1017.390,309.119,358.052,170.111,50.983,159.903
C03129=1017.397,309.366,358.020,170.117,50.978,159.903
C03130=1017.403,309.613,357.987,170.123,50.974,159.903
C03131=1017.410,309.861,357.954,170.129,50.970,159.903
C03132=1017.416,310.109,357.922,170.135,50.966,159.903
C03133=1017.422,310.356,357.889,170.141,50.961,159.903
C03134=1017.429,310.604,357.856,170.147,50.957,159.903
C03135=1017.435,310.852,357.822,170.153,50.953,159.903
C03136=1017.441,311.100,357.790,170.159,50.949,159.903
C03137=1017.447,311.348,357.757,170.165,50.945,159.903
C03138=1017.454,311.595,357.724,170.171,50.941,159.903
C03139=1017.460,311.842,357.691,170.177,50.937,159.903
C03140=1017.466,312.091,357.657,170.183,50.933,159.904
C03141=1017.473,312.338,357.624,170.189,50.928,159.904
C03142=1017.479,312.586,357.592,170.196,50.924,159.904
C03143=1017.486,312.833,357.558,170.202,50.920,159.904
C03144=1017.491,313.081,357.525,170.208,50.916,159.904
C03145=1017.498,313.329,357.492,170.214,50.912,159.904
C03146=1017.504,313.577,357.459,170.220,50.908,159.904
C03147=1017.511,313.824,357.425,170.227,50.904,159.905
C03148=1017.518,314.072,357.392,170.232,50.900,159.905
C03149=1017.523,314.320,357.359,170.239,50.896,159.905
C03150=1017.530,314.567,357.326,170.245,50.891,159.905
C03151=1017.536,314.814,357.293,170.251,50.888,159.905
C03152=1017.543,315.063,357.260,170.257,50.884,159.905
C03153=1017.550,315.310,357.226,170.263,50.880,159.905
C03154=1017.555,315.558,357.193,170.269,50.876,159.905
C03155=1017.562,315.805,357.159,170.275,50.872,159.906
C03156=1017.569,316.053,357.126,170.282,50.868,159.906
C03157=1017.576,316.301,357.093,170.287,50.864,159.906
C03158=1017.581,316.548,357.059,170.294,50.860,159.906
C03159=1017.588,316.795,357.026,170.300,50.856,159.906
C03160=1017.595,317.044,356.993,170.306,50.852,159.907
C03161=1017.602,317.291,356.959,170.313,50.848,159.907
C03162=1017.608,317.539,356.926,170.319,50.844,159.907
C03163=1017.614,317.786,356.892,170.325,50.840,159.907
C03164=1017.621,318.035,356.859,170.332,50.836,159.907
C03165=1017.628,318.281,356.825,170.338,50.833,159.907
C03166=1017.635,318.529,356.792,170.344,50.829,159.908
C03167=1017.641,318.777,356.758,170.350,50.825,159.908
C03168=1017.648,319.025,356.724,170.356,50.821,159.908
C03169=1017.654,319.272,356.692,170.363,50.818,159.908
C03170=1017.661,319.520,356.658,170.369,50.814,159.909
C03171=1017.668,319.768,356.624,170.375,50.810,159.909
C03172=1017.674,320.015,356.590,170.382,50.806,159.909
C03173=1017.681,320.263,356.557,170.389,50.802,159.909
C03174=1017.688,320.510,356.523,170.395,50.798,159.909
C03175=1017.695,320.758,356.490,170.401,50.795,159.910
C03176=1017.701,321.006,356.455,170.407,50.791,159.910
C03177=1017.708,321.253,356.422,170.414,50.787,159.910
C03178=1017.715,321.501,356.389,170.420,50.783,159.910
C03179=1017.722,321.749,356.355,170.426,50.780,159.910
C03180=1017.728,321.996,356.321,170.433,50.776,159.911
C03181=1017.736,322.258,356.286,170.439,50.772,159.911
C03182=1017.743,322.521,356.249,170.447,50.768,159.911
C03183=1017.750,322.783,356.213,170.453,50.764,159.911
C03184=1017.757,323.046,356.177,170.460,50.760,159.912
C03185=1017.764,323.293,356.144,170.467,50.757,159.912
C03186=1017.771,323.540,356.110,170.473,50.753,159.912
C03187=1017.778,323.788,356.076,170.479,50.749,159.913
C03188=1017.785,324.036,356.042,170.485,50.745,159.913
C03189=1017.792,324.284,356.008,170.493,50.741,159.913
C03190=1017.799,324.531,355.974,170.499,50.738,159.913
C03191=1017.806,324.778,355.941,170.506,50.734,159.914
C03192=1017.812,325.026,355.906,170.512,50.731,159.914
C03193=1017.819,325.274,355.873,170.518,50.728,159.914
C03194=1017.827,325.522,355.839,170.525,50.724,159.914
C03195=1017.833,325.769,355.804,170.532,50.720,159.915
C03196=1017.841,326.017,355.770,170.539,50.717,159.915
C03197=1017.848,326.264,355.736,170.545,50.713,159.915
C03198=1017.854,326.512,355.702,170.551,50.710,159.916
C03199=1017.861,326.759,355.667,170.558,50.706,159.916
C03200=1017.868,327.007,355.633,170.564,50.703,159.916
C03201=1017.874,327.254,355.598,170.570,50.699,159.917
C03202=1017.882,327.502,355.564,170.578,50.696,159.917
C03203=1017.888,327.749,355.529,170.585,50.693,159.918
C03204=1017.895,327.997,355.494,170.591,50.689,159.918
C03205=1017.902,328.244,355.459,170.598,50.686,159.918
C03206=1017.909,328.492,355.425,170.604,50.683,159.919
C03207=1017.916,328.739,355.390,170.610,50.679,159.919
C03208=1017.921,328.987,355.356,170.617,50.676,159.919
C03209=1017.929,329.234,355.322,170.625,50.672,159.920
C03210=1017.936,329.481,355.287,170.631,50.669,159.920
C03211=1017.942,329.729,355.252,170.638,50.666,159.920
C03212=1017.950,329.976,355.218,170.644,50.662,159.921
C03213=1017.956,330.223,355.183,170.651,50.659,159.921
C03214=1017.963,330.472,355.148,170.657,50.656,159.922
C03215=1017.970,330.720,355.113,170.664,50.652,159.922
C03216=1017.978,330.967,355.078,170.671,50.649,159.922
C03217=1017.984,331.214,355.043,170.678,50.646,159.923
C03218=1017.991,331.462,355.009,170.685,50.643,159.923
C03219=1017.998,331.709,354.974,170.691,50.640,159.923
C03220=1018.005,331.956,354.939,170.698,50.637,159.924
C03221=1018.012,332.204,354.904,170.705,50.633,159.924
C03222=1018.020,332.451,354.869,170.712,50.630,159.925
C03223=1018.026,332.698,354.834,170.719,50.627,159.925
C03224=1018.034,332.946,354.799,170.725,50.624,159.926
C03225=1018.040,333.194,354.763,170.732,50.621,159.926
C03226=1018.047,333.441,354.728,170.739,50.618,159.926
C03227=1018.054,333.688,354.693,170.746,50.614,159.927
C03228=1018.061,333.936,354.658,170.753,50.611,159.927
C03229=1018.067,334.183,354.623,170.759,50.608,159.928
C03230=1018.075,334.431,354.587,170.766,50.605,159.928
C03231=1018.082,334.678,354.552,170.773,50.602,159.928
C03232=1018.088,334.926,354.517,170.780,50.599,159.929
C03233=1018.095,335.173,354.481,170.787,50.596,159.930
C03234=1018.103,335.421,354.446,170.794,50.593,159.930
C03235=1018.110,335.668,354.411,170.801,50.590,159.930
C03236=1018.116,335.915,354.375,170.808,50.587,159.931
C03237=1018.123,336.162,354.340,170.814,50.584,159.931
C03238=1018.131,336.410,354.304,170.822,50.581,159.932
C03239=1018.138,336.658,354.269,170.828,50.578,159.932
C03240=1018.144,336.905,354.234,170.835,50.575,159.933
C03241=1018.152,337.163,354.197,170.843,50.572,159.933
C03242=1018.160,337.421,354.159,170.850,50.569,159.934
C03243=1018.167,337.679,354.122,170.858,50.566,159.935
C03244=1018.174,337.937,354.085,170.864,50.563,159.935
C03245=1018.182,338.185,354.050,170.871,50.560,159.935
C03246=1018.189,338.432,354.014,170.879,50.557,159.936
C03247=1018.196,338.679,353.979,170.886,50.554,159.936
C03248=1018.203,338.926,353.943,170.893,50.551,159.937
C03249=1018.210,339.174,353.907,170.899,50.548,159.937
C03250=1018.218,339.421,353.871,170.907,50.545,159.938
C03251=1018.225,339.668,353.835,170.914,50.542,159.939
C03252=1018.232,339.916,353.800,170.921,50.540,159.939
C03253=1018.239,340.163,353.763,170.928,50.537,159.940
C03254=1018.246,340.411,353.727,170.936,50.534,159.940
C03255=1018.253,340.657,353.691,170.943,50.532,159.941
C03256=1018.261,340.905,353.656,170.950,50.529,159.941
C03257=1018.268,341.152,353.620,170.956,50.526,159.942
C03258=1018.275,341.400,353.583,170.964,50.523,159.943
C03259=1018.282,341.647,353.547,170.971,50.521,159.943
C03260=1018.289,341.894,353.511,170.978,50.518,159.944
C03261=1018.296,342.141,353.475,170.985,50.515,159.944
C03262=1018.303,342.389,353.439,170.993,50.512,159.945
C03263=1018.311,342.637,353.403,171.000,50.510,159.945
C03264=1018.318,342.883,353.367,171.007,50.508,159.946
C03265=1018.326,343.131,353.331,171.015,50.505,159.947
C03266=1018.332,343.378,353.294,171.022,50.502,159.947
C03267=1018.340,343.625,353.258,171.029,50.499,159.948
C03268=1018.348,343.872,353.221,171.036,50.497,159.948
C03269=1018.354,344.119,353.185,171.044,50.494,159.949
C03270=1018.362,344.367,353.149,171.051,50.491,159.950
C03271=1018.369,344.614,353.112,171.058,50.489,159.950
C03272=1018.376,344.861,353.076,171.066,50.486,159.951
C03273=1018.383,345.109,353.040,171.073,50.484,159.952
C03274=1018.391,345.356,353.004,171.080,50.481,159.952
C03275=1018.398,345.603,352.966,171.088,50.479,159.953
C03276=1018.405,345.850,352.930,171.095,50.476,159.953
C03277=1018.413,346.097,352.894,171.102,50.474,159.954
C03278=1018.420,346.345,352.857,171.110,50.471,159.955
C03279=1018.428,346.592,352.820,171.117,50.469,159.956
C03280=1018.436,346.839,352.784,171.124,50.467,159.956
C03281=1018.442,347.087,352.747,171.132,50.464,159.957
C03282=1018.450,347.333,352.711,171.139,50.461,159.957
C03283=1018.457,347.581,352.674,171.147,50.459,159.958
C03284=1018.465,347.828,352.637,171.155,50.457,159.959
C03285=1018.472,348.076,352.600,171.162,50.454,159.960
C03286=1018.480,348.322,352.563,171.170,50.451,159.960
C03287=1018.487,348.570,352.526,171.177,50.450,159.961
C03288=1018.494,348.816,352.490,171.184,50.447,159.962
C03289=1018.501,349.063,352.452,171.192,50.445,159.963
C03290=1018.509,349.310,352.415,171.199,50.443,159.963
C03291=1018.516,349.558,352.378,171.206,50.440,159.964
C03292=1018.523,349.805,352.341,171.215,50.438,159.965
C03293=1018.531,350.052,352.304,171.222,50.435,159.965
C03294=1018.538,350.300,352.267,171.230,50.433,159.966
C03295=1018.546,350.547,352.230,171.237,50.431,159.967
C03296=1018.554,350.794,352.193,171.245,50.429,159.968
C03297=1018.561,351.041,352.155,171.253,50.426,159.968
C03298=1018.569,351.288,352.118,171.260,50.424,159.969
C03299=1018.576,351.535,352.081,171.268,50.422,159.970
C03300=1018.584,351.782,352.045,171.275,50.420,159.971
C03301=1018.592,352.038,352.006,171.284,50.418,159.972
C03302=1018.599,352.293,351.967,171.291,50.415,159.972
C03303=1018.608,352.548,351.928,171.299,50.413,159.973
C03304=1018.616,352.804,351.889,171.308,50.411,159.974
C03305=1018.623,353.051,351.852,171.315,50.409,159.975
C03306=1018.631,353.297,351.815,171.323,50.406,159.975
C03307=1018.638,353.545,351.777,171.331,50.404,159.976
C03308=1018.645,353.792,351.740,171.339,50.402,159.977
C03309=1018.653,354.039,351.703,171.346,50.400,159.978
C03310=1018.661,354.286,351.665,171.354,50.398,159.979
C03311=1018.669,354.534,351.628,171.362,50.396,159.979
C03312=1018.676,354.780,351.589,171.370,50.394,159.980
C03313=1018.684,355.027,351.552,171.378,50.392,159.981
C03314=1018.691,355.274,351.515,171.386,50.390,159.982
C03315=1018.699,355.521,351.476,171.393,50.388,159.983
C03316=1018.707,355.768,351.439,171.402,50.386,159.984
C03317=1018.714,356.016,351.401,171.409,50.384,159.985
C03318=1018.722,356.262,351.364,171.417,50.382,159.985
C03319=1018.730,356.510,351.326,171.425,50.380,159.986
C03320=1018.738,356.756,351.287,171.433,50.378,159.987
C03321=1018.745,357.003,351.250,171.441,50.376,159.988
C03322=1018.754,357.250,351.212,171.449,50.374,159.989
C03323=1018.761,357.497,351.174,171.456,50.372,159.990
C03324=1018.769,357.744,351.136,171.465,50.370,159.991
C03325=1018.776,357.992,351.098,171.473,50.368,159.992
C03326=1018.784,358.238,351.060,171.481,50.366,159.992
C03327=1018.792,358.485,351.021,171.488,50.364,159.993
C03328=1018.800,358.732,350.984,171.497,50.362,159.994
C03329=1018.808,358.979,350.946,171.506,50.361,159.995
C03330=1018.816,359.226,350.908,171.513,50.359,159.996
C03331=1018.824,359.473,350.869,171.521,50.357,159.997
C03332=1018.831,359.720,350.831,171.529,50.355,159.998
C03333=1018.839,359.967,350.793,171.538,50.353,159.999
C03334=1018.847,360.214,350.755,171.545,50.352,160.000
C03335=1018.854,360.461,350.716,171.554,50.350,160.001
C03336=1018.862,360.708,350.677,171.563,50.348,160.002
C03337=1018.869,360.955,350.639,171.570,50.346,160.003
C03338=1018.878,361.202,350.600,171.579,50.345,160.004
C03339=1018.886,361.449,350.562,171.586,50.343,160.005
C03340=1018.894,361.695,350.523,171.595,50.342,160.006
C03341=1018.902,361.942,350.484,171.603,50.339,160.007
C03342=1018.909,362.189,350.446,171.611,50.338,160.008
C03343=1018.917,362.436,350.407,171.620,50.337,160.009
C03344=1018.926,362.683,350.369,171.628,50.334,160.010
C03345=1018.932,362.930,350.330,171.636,50.333,160.011
C03346=1018.941,363.176,350.290,171.645,50.332,160.012
C03347=1018.949,363.424,350.252,171.653,50.329,160.013
C03348=1018.957,363.670,350.214,171.661,50.328,160.014
C03349=1018.965,363.917,350.174,171.670,50.327,160.015
C03350=1018.973,364.164,350.136,171.679,50.325,160.016
C03351=1018.981,364.410,350.097,171.686,50.323,160.017
C03352=1018.989,364.657,350.058,171.695,50.322,160.018
C03353=1018.997,364.904,350.020,171.703,50.320,160.019
C03354=1019.005,365.151,349.980,171.712,50.319,160.020
C03355=1019.013,365.398,349.941,171.720,50.317,160.021
C03356=1019.021,365.644,349.902,171.729,50.316,160.022
C03357=1019.029,365.892,349.863,171.738,50.314,160.023
C03358=1019.038,366.138,349.824,171.746,50.313,160.024
C03359=1019.046,366.385,349.785,171.754,50.312,160.025
C03360=1019.054,366.632,349.746,171.763,50.310,160.026
C03361=1019.062,366.895,349.705,171.772,50.308,160.027
C03362=1019.071,367.158,349.663,171.781,50.306,160.029
C03363=1019.081,367.420,349.621,171.790,50.305,160.030
C03364=1019.089,367.683,349.580,171.799,50.304,160.031
C03365=1019.097,367.930,349.540,171.808,50.302,160.032
C03366=1019.105,368.177,349.501,171.817,50.301,160.033
C03367=1019.113,368.424,349.461,171.826,50.299,160.034
C03368=1019.121,368.670,349.421,171.834,50.299,160.035
C03369=1019.129,368.917,349.382,171.843,50.297,160.037
C03370=1019.138,369.164,349.342,171.851,50.296,160.038
C03371=1019.145,369.411,349.302,171.861,50.295,160.039
C03372=1019.154,369.657,349.263,171.869,50.293,160.040
C03373=1019.162,369.904,349.224,171.878,50.291,160.041
C03374=1019.170,370.151,349.184,171.886,50.291,160.042
C03375=1019.179,370.397,349.144,171.895,50.289,160.043
C03376=1019.186,370.644,349.104,171.904,50.288,160.045
C03377=1019.195,370.890,349.064,171.913,50.287,160.046
C03378=1019.203,371.137,349.025,171.922,50.286,160.047
C03379=1019.212,371.384,348.984,171.931,50.284,160.048
C03380=1019.220,371.631,348.944,171.940,50.283,160.050
C03381=1019.228,371.877,348.905,171.949,50.282,160.051
C03382=1019.237,372.123,348.865,171.957,50.281,160.052
C03383=1019.245,372.370,348.825,171.966,50.280,160.053
C03384=1019.253,372.617,348.786,171.975,50.279,160.054
C03385=1019.262,372.864,348.745,171.984,50.278,160.056
C03386=1019.270,373.110,348.705,171.993,50.277,160.057
C03387=1019.278,373.357,348.665,172.003,50.276,160.058
C03388=1019.287,373.604,348.625,172.011,50.274,160.059
C03389=1019.295,373.850,348.584,172.020,50.273,160.061
C03390=1019.304,374.097,348.545,172.030,50.272,160.062
C03391=1019.313,374.343,348.505,172.039,50.271,160.063
C03392=1019.321,374.590,348.464,172.048,50.270,160.064
C03393=1019.330,374.836,348.425,172.057,50.269,160.066
C03394=1019.338,375.083,348.384,172.066,50.268,160.067
C03395=1019.347,375.329,348.344,172.075,50.267,160.068
C03396=1019.356,375.576,348.303,172.084,50.266,160.069
C03397=1019.364,375.823,348.263,172.093,50.265,160.071
C03398=1019.372,376.069,348.223,172.103,50.264,160.072
C03399=1019.381,376.316,348.182,172.113,50.263,160.074
C03400=1019.390,376.562,348.142,172.122,50.262,160.075
C03401=1019.398,376.809,348.101,172.131,50.261,160.076
C03402=1019.406,377.055,348.060,172.140,50.260,160.078
C03403=1019.415,377.302,348.019,172.150,50.259,160.079
C03404=1019.423,377.548,347.978,172.159,50.259,160.080
C03405=1019.433,377.795,347.937,172.168,50.258,160.082
C03406=1019.441,378.041,347.897,172.178,50.257,160.083
C03407=1019.449,378.288,347.856,172.187,50.256,160.084
C03408=1019.457,378.534,347.815,172.196,50.256,160.086
C03409=1019.466,378.781,347.773,172.205,50.255,160.087
C03410=1019.475,379.027,347.733,172.216,50.254,160.089
C03411=1019.484,379.274,347.692,172.225,50.253,160.090
C03412=1019.492,379.520,347.650,172.234,50.252,160.091
C03413=1019.500,379.766,347.610,172.244,50.252,160.093
C03414=1019.510,380.012,347.569,172.253,50.251,160.094
C03415=1019.519,380.259,347.528,172.262,50.250,160.096
C03416=1019.527,380.505,347.486,172.273,50.250,160.097
C03417=1019.536,380.752,347.445,172.282,50.249,160.099
C03418=1019.545,380.998,347.404,172.292,50.248,160.100
C03419=1019.554,381.245,347.363,172.301,50.247,160.101
C03420=1019.563,381.491,347.322,172.311,50.247,160.103
C03421=1019.573,381.776,347.274,172.322,50.246,160.105
C03422=1019.583,382.061,347.226,172.334,50.245,160.106
C03423=1019.593,382.346,347.178,172.344,50.245,160.108
C03424=1019.604,382.631,347.131,172.356,50.244,160.110
C03425=1019.613,382.877,347.089,172.365,50.243,160.111
C03426=1019.622,383.124,347.047,172.376,50.242,160.113
C03427=1019.631,383.371,347.006,172.386,50.242,160.114
C03428=1019.639,383.617,346.965,172.395,50.242,160.116
C03429=1019.649,383.863,346.924,172.406,50.241,160.117
C03430=1019.658,384.109,346.882,172.415,50.241,160.119
C03431=1019.667,384.355,346.840,172.425,50.240,160.121
C03432=1019.675,384.602,346.799,172.435,50.239,160.122
C03433=1019.685,384.849,346.756,172.445,50.239,160.124
C03434=1019.695,385.095,346.715,172.455,50.238,160.125
C03435=1019.704,385.341,346.674,172.465,50.238,160.127
C03436=1019.713,385.587,346.631,172.474,50.238,160.128
C03437=1019.722,385.833,346.589,172.485,50.237,160.130
C03438=1019.731,386.080,346.548,172.495,50.237,160.132
C03439=1019.740,386.326,346.506,172.505,50.236,160.133
C03440=1019.748,386.572,346.463,172.515,50.236,160.135
C03441=1019.757,386.818,346.421,172.525,50.235,160.136
C03442=1019.766,387.064,346.379,172.535,50.235,160.138
C03443=1019.776,387.311,346.337,172.546,50.235,160.140
C03444=1019.785,387.557,346.294,172.556,50.235,160.141
C03445=1019.794,387.803,346.253,172.566,50.234,160.143
C03446=1019.803,388.049,346.210,172.576,50.234,160.145
C03447=1019.813,388.296,346.168,172.587,50.234,160.146
C03448=1019.822,388.542,346.126,172.597,50.234,160.148
C03449=1019.831,388.788,346.083,172.607,50.233,160.150
C03450=1019.840,389.034,346.040,172.617,50.233,160.151
C03451=1019.849,389.281,345.998,172.628,50.233,160.153
C03452=1019.859,389.526,345.956,172.638,50.233,160.155
C03453=1019.868,389.772,345.913,172.649,50.232,160.156
C03454=1019.878,390.019,345.871,172.660,50.232,160.158
C03455=1019.886,390.265,345.827,172.669,50.232,160.160
C03456=1019.896,390.511,345.785,172.680,50.232,160.161
C03457=1019.905,390.757,345.742,172.691,50.232,160.163
C03458=1019.914,391.003,345.700,172.701,50.232,160.165
C03459=1019.924,391.249,345.657,172.712,50.232,160.167
C03460=1019.933,391.495,345.614,172.723,50.231,160.169
C03461=1019.943,391.742,345.571,172.733,50.232,160.170
C03462=1019.952,391.987,345.529,172.744,50.231,160.172
C03463=1019.962,392.234,345.486,172.754,50.231,160.174
C03464=1019.972,392.480,345.442,172.764,50.231,160.176
C03465=1019.980,392.726,345.399,172.775,50.231,160.177
C03466=1019.990,392.972,345.357,172.786,50.231,160.179
C03467=1019.999,393.218,345.313,172.797,50.231,160.181
C03468=1020.009,393.464,345.270,172.807,50.231,160.183
C03469=1020.018,393.709,345.227,172.818,50.232,160.185
C03470=1020.028,393.956,345.184,172.829,50.231,160.187
C03471=1020.038,394.202,345.140,172.840,50.231,160.188
C03472=1020.047,394.447,345.098,172.852,50.232,160.190
C03473=1020.056,394.694,345.053,172.861,50.232,160.192
C03474=1020.066,394.939,345.010,172.872,50.232,160.194
C03475=1020.076,395.186,344.967,172.884,50.232,160.196
C03476=1020.085,395.431,344.923,172.895,50.232,160.198
C03477=1020.095,395.677,344.880,172.906,50.232,160.200
C03478=1020.105,395.923,344.836,172.917,50.232,160.202
C03479=1020.115,396.170,344.793,172.928,50.232,160.204
C03480=1020.124,396.416,344.749,172.939,50.232,160.205
C03481=1020.137,396.738,344.692,172.953,50.233,160.208
C03482=1020.150,397.060,344.635,172.968,50.233,160.211
C03483=1020.162,397.383,344.577,172.983,50.234,160.213
C03484=1020.176,397.705,344.520,172.998,50.234,160.216
C03485=1020.185,397.951,344.475,173.009,50.234,160.218
C03486=1020.196,398.197,344.432,173.020,50.234,160.220
C03487=1020.205,398.443,344.388,173.032,50.235,160.222
C03488=1020.215,398.689,344.343,173.043,50.235,160.224
C03489=1020.225,398.935,344.300,173.054,50.235,160.226
C03490=1020.234,399.181,344.255,173.065,50.236,160.228
C03491=1020.245,399.426,344.211,173.077,50.236,160.230
C03492=1020.254,399.672,344.167,173.088,50.237,160.232
C03493=1020.264,399.918,344.122,173.099,50.237,160.234
C03494=1020.274,400.163,344.079,173.112,50.237,160.236
C03495=1020.284,400.409,344.034,173.123,50.237,160.238
C03496=1020.294,400.655,343.990,173.134,50.238,160.240
C03497=1020.304,400.901,343.945,173.146,50.239,160.242
C03498=1020.314,401.146,343.900,173.157,50.239,160.244
C03499=1020.323,401.393,343.856,173.169,50.240,160.246
C03500=1020.333,401.638,343.811,173.181,50.240,160.249
C03501=1020.343,401.883,343.767,173.193,50.240,160.251
C03502=1020.354,402.130,343.722,173.204,50.241,160.253
C03503=1020.363,402.375,343.677,173.216,50.242,160.255
C03504=1020.373,402.621,343.632,173.228,50.242,160.257
C03505=1020.384,402.866,343.588,173.240,50.243,160.259
C03506=1020.394,403.112,343.543,173.251,50.244,160.262
C03507=1020.404,403.357,343.498,173.263,50.244,160.264
C03508=1020.414,403.604,343.453,173.275,50.245,160.266
C03509=1020.424,403.849,343.408,173.287,50.246,160.268
C03510=1020.435,404.095,343.364,173.299,50.246,160.270
C03511=1020.445,404.340,343.318,173.311,50.247,160.272
C03512=1020.455,404.586,343.273,173.323,50.247,160.275
C03513=1020.465,404.832,343.228,173.335,50.248,160.277
C03514=1020.475,405.077,343.182,173.347,50.249,160.279
C03515=1020.486,405.323,343.138,173.360,50.250,160.282
C03516=1020.496,405.569,343.093,173.371,50.251,160.284
C03517=1020.507,405.814,343.047,173.384,50.251,160.286
C03518=1020.517,406.060,343.002,173.396,50.252,160.288
C03519=1020.527,406.305,342.956,173.409,50.253,160.291
C03520=1020.538,406.551,342.911,173.420,50.253,160.293
C03521=1020.549,406.797,342.866,173.433,50.254,160.295
C03522=1020.559,407.042,342.820,173.445,50.255,160.297
C03523=1020.569,407.288,342.775,173.457,50.256,160.300
C03524=1020.581,407.533,342.729,173.470,50.256,160.302
C03525=1020.591,407.779,342.684,173.482,50.258,160.305
C03526=1020.602,408.025,342.638,173.495,50.258,160.307
C03527=1020.612,408.270,342.593,173.507,50.259,160.309
C03528=1020.622,408.516,342.547,173.520,50.260,160.312
C03529=1020.634,408.761,342.502,173.532,50.261,160.314
C03530=1020.644,409.007,342.456,173.545,50.262,160.316
C03531=1020.655,409.252,342.410,173.557,50.263,160.319
C03532=1020.665,409.498,342.363,173.570,50.264,160.321
C03533=1020.675,409.744,342.317,173.583,50.264,160.324
C03534=1020.686,409.989,342.271,173.596,50.266,160.326
C03535=1020.697,410.234,342.225,173.608,50.267,160.329
C03536=1020.707,410.480,342.179,173.621,50.268,160.331
C03537=1020.718,410.725,342.132,173.634,50.269,160.333
C03538=1020.730,410.971,342.086,173.647,50.270,160.336
C03539=1020.740,411.217,342.040,173.660,50.271,160.338
C03540=1020.751,411.462,341.994,173.673,50.272,160.341
C03541=1020.766,411.807,341.928,173.690,50.274,160.344
C03542=1020.781,412.153,341.863,173.709,50.276,160.348
C03543=1020.797,412.498,341.798,173.727,50.277,160.352
C03544=1020.811,412.843,341.732,173.746,50.278,160.355
C03545=1020.823,413.088,341.685,173.760,50.280,160.358
C03546=1020.834,413.333,341.638,173.773,50.281,160.361
C03547=1020.845,413.579,341.592,173.786,50.282,160.363
C03548=1020.856,413.824,341.545,173.799,50.283,160.366
C03549=1020.867,414.069,341.498,173.812,50.285,160.368
C03550=1020.878,414.316,341.451,173.826,50.286,160.371
C03551=1020.889,414.561,341.405,173.839,50.287,160.374
C03552=1020.901,414.806,341.357,173.852,50.289,160.376
C03553=1020.912,415.051,341.310,173.866,50.290,160.379
C03554=1020.923,415.296,341.263,173.880,50.291,160.382
C03555=1020.934,415.542,341.216,173.893,50.293,160.384
C03556=1020.945,415.787,341.169,173.907,50.294,160.387
C03557=1020.956,416.033,341.121,173.920,50.295,160.390
C03558=1020.967,416.278,341.074,173.933,50.297,160.392
C03559=1020.979,416.523,341.027,173.948,50.298,160.395
C03560=1020.989,416.769,340.979,173.961,50.300,160.398
C03561=1021.001,417.013,340.932,173.975,50.301,160.401
C03562=1021.012,417.259,340.885,173.989,50.303,160.404
C03563=1021.023,417.504,340.836,174.003,50.304,160.406
C03564=1021.035,417.749,340.789,174.016,50.306,160.409
C03565=1021.045,417.994,340.742,174.030,50.307,160.412
C03566=1021.057,418.239,340.694,174.044,50.309,160.415
C03567=1021.069,418.484,340.646,174.058,50.310,160.418
C03568=1021.080,418.730,340.598,174.072,50.312,160.420
C03569=1021.092,418.975,340.550,174.087,50.313,160.423
C03570=1021.104,419.220,340.502,174.100,50.315,160.426
C03571=1021.115,419.465,340.454,174.115,50.316,160.429
C03572=1021.127,419.710,340.406,174.129,50.318,160.432
C03573=1021.139,419.955,340.359,174.143,50.320,160.435
C03574=1021.150,420.201,340.310,174.158,50.321,160.438
C03575=1021.161,420.446,340.263,174.171,50.323,160.441
C03576=1021.173,420.691,340.214,174.186,50.325,160.444
C03577=1021.185,420.936,340.166,174.201,50.326,160.446
C03578=1021.197,421.181,340.118,174.215,50.328,160.449
C03579=1021.208,421.427,340.070,174.229,50.330,160.453
C03580=1021.220,421.671,340.021,174.244,50.331,160.455
C03581=1021.231,421.916,339.973,174.259,50.333,160.458
C03582=1021.243,422.161,339.924,174.273,50.335,160.461
C03583=1021.255,422.406,339.875,174.287,50.337,160.464
C03584=1021.267,422.652,339.827,174.302,50.338,160.467
C03585=1021.279,422.896,339.778,174.317,50.340,160.471
C03586=1021.290,423.141,339.729,174.332,50.342,160.474
C03587=1021.302,423.386,339.680,174.347,50.344,160.477
C03588=1021.314,423.631,339.632,174.362,50.346,160.480
C03589=1021.326,423.877,339.583,174.377,50.348,160.483
C03590=1021.338,424.121,339.534,174.392,50.349,160.486
C03591=1021.350,424.365,339.485,174.407,50.351,160.489
C03592=1021.363,424.610,339.436,174.422,50.354,160.492
C03593=1021.375,424.856,339.387,174.437,50.355,160.495
C03594=1021.386,425.101,339.338,174.452,50.358,160.499
C03595=1021.399,425.346,339.289,174.467,50.359,160.502
C03596=1021.411,425.591,339.239,174.482,50.362,160.505
C03597=1021.423,425.835,339.190,174.498,50.363,160.508
C03598=1021.435,426.081,339.140,174.513,50.365,160.511
C03599=1021.446,426.325,339.091,174.529,50.367,160.515
C03600=1021.459,426.570,339.042,174.544,50.370,160.518
C03601=1021.471,426.810,338.993,174.559,50.371,160.521
C03602=1021.483,427.050,338.944,174.574,50.374,160.524
C03603=1021.495,427.290,338.896,174.589,50.376,160.528
C03604=1021.507,427.530,338.847,174.605,50.378,160.531
C03605=1021.519,427.770,338.798,174.620,50.379,160.534
C03606=1021.531,428.009,338.748,174.636,50.382,160.537
C03607=1021.544,428.249,338.700,174.651,50.384,160.541
C03608=1021.555,428.488,338.651,174.666,50.386,160.544
C03609=1021.567,428.733,338.601,174.682,50.388,160.547
C03610=1021.580,428.978,338.551,174.698,50.391,160.551
C03611=1021.592,429.223,338.501,174.714,50.393,160.554
C03612=1021.605,429.467,338.451,174.730,50.395,160.557
C03613=1021.618,429.712,338.401,174.746,50.397,160.561
C03614=1021.630,429.956,338.351,174.762,50.399,160.564
C03615=1021.643,430.202,338.300,174.778,50.402,160.568
C03616=1021.655,430.446,338.249,174.795,50.404,160.571
C03617=1021.272,428.491,338.315,174.655,50.455,160.562
C03618=1021.261,428.264,338.361,174.641,50.453,160.559
C03619=1021.250,428.037,338.408,174.626,50.451,160.556
C03620=1021.238,427.810,338.453,174.611,50.449,160.553
C03621=1021.227,427.582,338.500,174.597,50.447,160.550
C03622=1021.216,427.356,338.546,174.582,50.445,160.547
C03623=1021.204,427.128,338.592,174.567,50.444,160.544
C03624=1021.193,426.901,338.639,174.553,50.442,160.541
C03625=1021.182,426.673,338.685,174.539,50.440,160.538
C03626=1021.169,426.429,338.733,174.523,50.438,160.534
C03627=1021.157,426.184,338.784,174.508,50.436,160.531
C03628=1021.146,425.939,338.833,174.492,50.434,160.528
C03629=1021.133,425.695,338.883,174.477,50.432,160.525
C03630=1021.121,425.449,338.932,174.462,50.430,160.522
C03631=1021.109,425.205,338.980,174.447,50.428,160.518
C03632=1021.097,424.959,339.030,174.431,50.426,160.515
